      A     DB210.DBX  988.0;
      A     DB210.DBX  982.6;
      S     DB115.DBX   26.4;
      JCN   AFrm;
      L     #ComLine;
      L     128;
      OW    ;
      T     #ComLine;
AFrm: NOP   0;

//Frischwasser
      A     DB1565.DBX   26.1;
      A     #ComU056;
      A     M    103.3;
      =     DB210.DBX  108.0;

      A     DB210.DBX  108.0;
      A     DB210.DBX  102.6;
      S     DB115.DBX   26.4;
      JCN   AXrm;
      L     #ComLine;
      L     256;
      OW    ;
      T     #ComLine;
AXrm: NOP   0;

//Brauhaus
      A     DB1575.DBX   26.1;
      A     #ComU057;
      A     M    103.3;
      =     DB210.DBX  188.0;

      A     DB210.DBX  188.0;
      A     DB210.DBX  182.6;
      S     DB115.DBX   26.4;
      JCN   AYrm;
      L     #ComLine;
      L     512;
      OW    ;
      T     #ComLine;
AYrm: NOP   0;
//Sirupraum
      A     DB1585.DBX   26.1;
      A     #ComU058;
      A     M    103.3;
      =     DB210.DBX  348.0;

      A     DB210.DBX  348.0;
      A     DB210.DBX  342.6;
      S     DB115.DBX   26.4;
      JCN   AZrm;
      L     #ComLine;
      L     1024;
      OW    ;
      T     #ComLine;
AZrm: NOP   0;


      A     #ComSRC;
      A     DB115.DBX  218.4;
      A     M    103.3;
      =     #ReqInlet;

// -------------------------------------------------
// subphase transition
      AN    #reqAnlage;
      AN    DB115.DBX  218.4;
      =     M    103.1;
      JU    COMM;
NETWORK
TITLE =phase 8: Emptying
//SFM   Use                                 Datatype        UoM
//----+-------------------------------------------------------------------------
// 00 : Watch Dog Time                      Duration        min
// 04 : Delay Empty                         Duration        s
// 17 : Level                               Value           l
X8:   SET   ;
// ---------------------------------------------------------------------------
// General CM evaluation
      CALL FC   110 (
           ChkType                  := 3,
           ChkOK                    := #ChkOK);

      AN    #ChkOK;
      S     M    120.3;

// ---------------------------------------------------------------------------
// general functions
      AN    M    121.2;
      A     M    102.3;
      =     #RRel;

      A     M    102.3;
      S     DB115.DBX   26.3;

      A     M    152.1; // Befüllfreigabe
      A     M    102.3;
      S     DB115.DBX   26.0;

// ---------------------------------------------------------------------------
// messages
// ---------------------------------------------------------------------------
// timer & counter

// ---------------------------------------------------------------------------
// pause timer
      ON    M    102.3;
      O     M    150.3;
      S     M    140.3; // Delay Empty

// ---------------------------------------------------------------------------
// communication
      A     DB1435.DBX   26.1;
      A     #ComU043;
      O     ;
      A     DB1455.DBX   26.1;
      A     #ComU045;
      O     ;
      A     DB1475.DBX   26.1;
      A     #ComU047;
      O     ;
      A     DB1485.DBX   26.1;
      A     #ComU048;
      O     ;
      A     DB1495.DBX   26.1;
      A     #ComU049;
      O     ;
      A     DB1505.DBX   26.1;
      A     #ComU050;
      O     ;
      A     DB1515.DBX   26.1;
      A     #ComU051;
      O     ;
      A     DB1525.DBX   26.1;
      A     #ComU052;
      O     ;
      A     DB1545.DBX   26.1;
      A     #ComU054;
      O     ;
      A     DB1555.DBX   26.1;
      A     #ComU055;
      O     ;
      A     DB1565.DBX   26.1;
      A     #ComU056;
      O     ;
      A     DB1575.DBX   26.1;
      A     #ComU057;
      O     ;
      A     DB1585.DBX   26.1;
      A     #ComU058;
      =     #reqAnlage;


// ---------------------------------------------------------------------------
// control modules
      A     M    102.3;

// ---------------------------------------------------------------------------
// transition condition
      A     #U.Seq.User.Bit5; // FILL_REL
      A     DB115.DBX  218.3;
      AN    M    102.2;
      =     M    102.1;
      JCN   N501;
      L     MW   104;
      L     1; // Return to Production
      -I    ;
      T     MW   106;
N501: NOP   0;

      AN    #U.Seq.User.Bit6; // EMPTY_REL
      A     #U.Seq.User.Bit5; // FILL_REL
      AN    M    102.2;
      S     M    102.1;
      JCN   N502;
      L     MW   104;
      L     2; // Return to Filling
      -I    ;
      T     MW   106;
N502: NOP   0;


// ---------------------------------------------------------------------------
// ---------------------------------------------------------------------------
// subphase repeat function
      A     #SubStepMax;
      JCN   Y8;
      L     1;
      T     MW   116;
Y8:   SET   ;

// subphase evaluation
      L     MW   110;
      JL    A800;
      JU    COMM; // subphase  0:
      JU    A801; // subphase  1: Waiting
      JU    A802; // subphase  2: Active
// ---------------------------------------------------------------------------
A800: SET   ;
      S     M    110.7; // Error unknown subphase
      JU    COMM;

// subphase 1: Waiting
A801: SET   ;
      A     M    103.0;
      R     DB115.DBX   26.4;
// -------------------------------------------------
// subphase timer & counter
      A     M    103.0;

// -------------------------------------------------
// subphase actuator
      A     M    103.3;

// -------------------------------------------------
// subphase transition
      A     #reqAnlage;
//      AN    "C01SpiD".LABOR_FREIG_T13.Sig
      =     M    103.1;
      JU    COMM;

// subphase 2: Active
A802: SET   ;
      A     M    103.0;
      =     DB115.DBX   26.4;
// -------------------------------------------------
// subphase timer & counter
      A     M    103.0;

// -------------------------------------------------
// subphase actuator
// Emptying -------------
      CLR   ;
      =     DB115.DBX   26.4;
//KEG
      A     DB1435.DBX   26.1;
      A     #ComU043;
      A     M    103.3;
      =     DB210.DBX  268.0;

      A     DB210.DBX  268.0;
      A     DB210.DBX  262.6;
      S     DB115.DBX   26.4;
      JCN   A3rn;
      L     #ComLine;
      L     1;
      OW    ;
      T     #ComLine;
A3rn: NOP   0;
//A5
      A     DB1455.DBX   26.1;
      A     #ComU045;
      A     M    103.3;
      =     DB210.DBX  828.0;

      A     DB210.DBX  828.0;
      A     DB210.DBX  822.6;
      S     DB115.DBX   26.4;
      JCN   A5rn;
      L     #ComLine;
      L     2;
      OW    ;
      T     #ComLine;
A5rn: NOP   0;

//A7
      A     DB1475.DBX   26.1;
      A     #ComU047;
      A     M    103.3;
      =     DB210.DBX  668.0;

      A     DB210.DBX  668.0;
      A     DB210.DBX  662.6;
      S     DB115.DBX   26.4;
      JCN   A7rn;
      L     #ComLine;
      L     4;
      OW    ;
      T     #ComLine;
A7rn: NOP   0;

//A9
      A     DB1495.DBX   26.1;
      A     #ComU049;
      A     M    103.3;
      =     DB210.DBX  508.0;

      A     DB210.DBX  508.0;
      A     DB210.DBX  502.6;
      S     DB115.DBX   26.4;
      JCN   A9rn;
      L     #ComLine;
      L     8;
      OW    ;
      T     #ComLine;
A9rn: NOP   0;

//A10
      A     DB1505.DBX   26.1;
      A     #ComU050;
      A     M    103.3;
      =     DB210.DBX  428.0;

      A     DB210.DBX  428.0;
      A     DB210.DBX  422.6;
      S     DB115.DBX   26.4;
      JCN   AArn;
      L     #ComLine;
      L     16;
      OW    ;
      T     #ComLine;
AArn: NOP   0;

//A11
      A     DB1515.DBX   26.1;
      A     #ComU051;
      A     M    103.3;
      =     DB210.DBX  908.0;

      A     DB210.DBX  908.0;
      A     DB210.DBX  902.6;
      S     DB115.DBX   26.4;
      JCN   ABrn;
      L     #ComLine;
      L     32;
      OW    ;
      T     #ComLine;
ABrn: NOP   0;

//A12
      A     DB1525.DBX   26.1;
      A     #ComU052;
      A     M    103.3;
      =     DB210.DBX  588.0;

      A     DB210.DBX  588.0;
      A     DB210.DBX  582.6;
      S     DB115.DBX   26.4;
      JCN   ACrn;
      L     #ComLine;
      L     64;
      OW    ;
      T     #ComLine;
ACrn: NOP   0;

//A14
      A     DB1545.DBX   26.1;
      A     #ComU054;
      A     M    103.3;
      =     DB210.DBX  988.0;

      A     DB210.DBX  988.0;
      A     DB210.DBX  982.6;
      S     DB115.DBX   26.4;
      JCN   AFrn;
      L     #ComLine;
      L     128;
      OW    ;
      T     #ComLine;
AFrn: NOP   0;

//Frischwasser
      A     DB1565.DBX   26.1;
      A     #ComU056;
      A     M    103.3;
      =     DB210.DBX  108.0;

      A     DB210.DBX  108.0;
      A     DB210.DBX  102.6;
      S     DB115.DBX   26.4;
      JCN   AXrn;
      L     #ComLine;
      L     256;
      OW    ;
      T     #ComLine;
AXrn: NOP   0;

//Brauhaus
      A     DB1575.DBX   26.1;
      A     #ComU057;
      A     M    103.3;
      =     DB210.DBX  188.0;

      A     DB210.DBX  188.0;
      A     DB210.DBX  182.6;
      S     DB115.DBX   26.4;
      JCN   AYrn;
      L     #ComLine;
      L     512;
      OW    ;
      T     #ComLine;
AYrn: NOP   0;
//Sirupraum
      A     DB1585.DBX   26.1;
      A     #ComU058;
      A     M    103.3;
      =     DB210.DBX  348.0;

      A     DB210.DBX  348.0;
      A     DB210.DBX  342.6;
      S     DB115.DBX   26.4;
      JCN   AZrn;
      L     #ComLine;
      L     1024;
      OW    ;
      T     #ComLine;
AZrn: NOP   0;


// -------------------------------------------------
// subphase transition
      AN    #reqAnlage;
      =     M    103.1;
      JU    COMM;
NETWORK
TITLE =phase 20: Quality Check
//SFM   Use                                 Datatype        UoM
//----+-------------------------------------------------------------------------
// 00 : Watch Dog Time                      Duration        min
// 39 : Q-Status                            Enumeration     min
X20:  SET   ;
// ---------------------------------------------------------------------------
// General CM evaluation
      CALL FC   110 (
           ChkType                  := 3,
           ChkOK                    := #ChkOK);

      AN    #ChkOK;
      S     M    120.3;

// ---------------------------------------------------------------------------
// index evaluation: Q-Status
      CALL FC    45 (
           SFM                      := #U.Seq.SFM[39].Sp,
           Indexes                  := #S2I.SFM39);

// ---------------------------------------------------------------------------
// general functions
      AN    M    121.2;
      A     M    102.3;
      =     #RRel;

// ---------------------------------------------------------------------------
// messages
// ---------------------------------------------------------------------------
// timer & counter
      A     M    102.0;

// ---------------------------------------------------------------------------
// pause timer
// ---------------------------------------------------------------------------
// communication

// ---------------------------------------------------------------------------
// control modules
      A     M    102.3;

// ---------------------------------------------------------------------------
// transition condition
      A     #SubStepMaxD;
      =     M    102.1;

// subphase evaluation
      L     MW   110;
      JL    C000;
      JU    COMM; // subphase  0:
// ---------------------------------------------------------------------------
C000: SET   ;
      S     M    110.7; // Error unknown subphase
      JU    COMM;
NETWORK
TITLE =phase 21: Prepare Tank
//SFM   Use                                 Datatype        UoM
//----+-------------------------------------------------------------------------
// 00 : Watch Dog Time                      Duration        min
// 17 : Level                               Value           l
X21:  SET   ;
// ---------------------------------------------------------------------------
// General CM evaluation
      CALL FC   110 (
           ChkType                  := 3,
           ChkOK                    := #ChkOK);

      AN    #ChkOK;
      S     M    120.3;

// ---------------------------------------------------------------------------
// general functions
      AN    M    121.2;
      A     M    102.3;
      =     #RRel;

// ---------------------------------------------------------------------------
// messages
// ---------------------------------------------------------------------------
// timer & counter
      A     M    102.0;

// ---------------------------------------------------------------------------
// pause timer
// ---------------------------------------------------------------------------
// communication

// ---------------------------------------------------------------------------
// control modules

      CLR   ;
      =     DB211.DBX  503.1; // Filling Hand Valve
      =     DB211.DBX  623.1; // CIP Hand Valve

      A     M    102.3;
      =     DB211.DBX  503.0; // Filling Hand Valve
      =     DB211.DBX  623.0; // CIP Hand Valve

// ---------------------------------------------------------------------------
// transition condition
      AN    DB211.DBX  498.7; // Filling Hand Valve
      AN    DB211.DBX  618.7; // CIP Hand Valve
      AN    M    102.2;
      =     M    102.1;

// subphase evaluation
      L     MW   110;
      JL    C100;
      JU    COMM; // subphase  0:
// ---------------------------------------------------------------------------
C100: SET   ;
      S     M    110.7; // Error unknown subphase
      JU    COMM;
NETWORK
TITLE =phase 23: Connect Tank
//SFM   Use                                 Datatype        UoM
//----+-------------------------------------------------------------------------
// 00 : Watch Dog Time                      Duration        min
X23:  SET   ;
// ---------------------------------------------------------------------------
// General CM evaluation
      CALL FC   110 (
           ChkType                  := 3,
           ChkOK                    := #ChkOK);

      AN    #ChkOK;
      S     M    120.3;

// ---------------------------------------------------------------------------
// general functions
      AN    M    121.2;
      A     M    102.3;
      =     #RRel;

// ---------------------------------------------------------------------------
// messages
// ---------------------------------------------------------------------------
// timer & counter
      A     M    102.0;

// ---------------------------------------------------------------------------
// pause timer
// ---------------------------------------------------------------------------
// communication

// ---------------------------------------------------------------------------
// control modules
      A     M    102.3;

// ---------------------------------------------------------------------------
// transition condition
      A     #SubStepMaxD;
      =     M    102.1;

// subphase evaluation
      L     MW   110;
      JL    C300;
      JU    COMM; // subphase  0:
// ---------------------------------------------------------------------------
C300: SET   ;
      S     M    110.7; // Error unknown subphase
      JU    COMM;
NETWORK
TITLE =phase 31: CIP Start
//SFM   Use                                 Datatype        UoM
//----+-------------------------------------------------------------------------
// 00 : Watch Dog Time                      Duration        min
X31:  SET   ;
// ---------------------------------------------------------------------------
// General CM evaluation
      CALL FC   110 (
           ChkType                  := 4,
           ChkOK                    := #ChkOK);

      AN    #ChkOK;
      S     M    120.3;

// ---------------------------------------------------------------------------
// general functions
      AN    M    121.2;
      A     M    102.3;
      =     #RRel;

// ---------------------------------------------------------------------------
// messages
// ---------------------------------------------------------------------------
// timer & counter
// ---------------------------------------------------------------------------
// pause timer
// ---------------------------------------------------------------------------
// communication

// ---------------------------------------------------------------------------
// control modules

// ---------------------------------------------------------------------------
// transition condition
      A     #SubStepMaxD;
      =     M    102.1;

// ---------------------------------------------------------------------------
// ---------------------------------------------------------------------------
// subphase repeat function
//      A     #SubStepMax
//      JCN  Y31
//      L     1
//      T     "SOSubStepNew"
//Y31:  SET

// subphase evaluation
      L     MW   110;
      JL    D100;
      JU    COMM; // subphase  0:
      JU    D101; // subphase  1: Wait For CIP
      JU    D102; // subphase  2: Wait For Partner
// ---------------------------------------------------------------------------
D100: SET   ;
      S     M    110.7; // Error unknown subphase
      JU    COMM;

// subphase 1: Wait For CIP
D101: SET   ;

// -------------------------------------------------
// CIP Signals ---
// Start Signal
      A     M    120.0;
      A     M    103.3;
      =     DB115.DBX  172.4;
      JCN   CIPS;
      L     MD   124;
      T     DB502.DBD    0;
      T     DB502.DBD  156;
CIPS: NOP   0;

// -------------------------------------------------
// subphase actuator

// -------------------------------------------------
// subphase transition
// CIP Ready
      A     #ComCIP;
      A     DB115.DBX  123.5;
      A     DB115.DBX  120.0;
// CIP Distribution Ready
      A     #ComCIPDist;
      A     DB1945.DBX   27.5;
      A     DB1945.DBX   24.0;
      =     M    103.1;
      JU    COMM;

// subphase 2: Wait For Partner
D102: SET   ;

// -------------------------------------------------
// subphase timer & counter
      A     M    103.0;

// -------------------------------------------------
// subphase actuator
      A     M    103.3;

// -------------------------------------------------
// subphase transition
      CLR   ;
      =     M    103.1;
      JU    COMM;
NETWORK
TITLE =phase 32: CIP Prerun
//SFM   Use                                 Datatype        UoM
//----+-------------------------------------------------------------------------
// 00 : Watch Dog Time                      Duration        min
// 01 : Step Time                           Duration        min
// 04 : Delay Level                         Duration        s
// 15 : Amount                              Value           m3
// 17 : Level                               Value           l
// 22 : Agitator Speed                      Value           %
// 27 : CIP Prerun                          Enumeration     min
// 28 : CIP Return                          Enumeration     min
// 29 : CIP Pump Speed                      Value           %
// 34 : CIP Prerun Flow                     Value           m3/h
// 35 : CIP Prerun Pressure                 Value           bar
// 37 : CIP Pump Mode                       Enumeration     min
X32:  SET   ;
// ---------------------------------------------------------------------------
// General CM evaluation
      CALL FC   110 (
           ChkType                  := 4,
           ChkOK                    := #ChkOK);

      AN    #ChkOK;
      S     M    120.3;

// ---------------------------------------------------------------------------
// index evaluation: CIP Prerun
      CALL FC    45 (
           SFM                      := #U.Seq.SFM[27].Sp,
           Indexes                  := #S2I.SFM27);

// ---------------------------------------------------------------------------
// index evaluation: CIP Return
      CALL FC    45 (
           SFM                      := #U.Seq.SFM[28].Sp,
           Indexes                  := #S2I.SFM28);

// ---------------------------------------------------------------------------
// index evaluation: CIP Pump Mode
      CALL FC    45 (
           SFM                      := #U.Seq.SFM[37].Sp,
           Indexes                  := #S2I.SFM37);

// ---------------------------------------------------------------------------
// general functions
      AN    M    121.2;
      A     M    102.3;
      =     #RRel;

// ---------------------------------------------------------------------------
// messages
// CIP Unit
      AN    #ComCIP;
      ON    DB115.DBX  123.4;
      ON    DB115.DBX  123.5;
      JCN   x321;
      R     #RRel;
      L     949; // CIP Not Ready!
      T     MD    90;
x321: NOP   0;

// CIP Distribution Unit
      AN    #ComCIPDist;
      ON    DB1945.DBX   27.4;
      ON    DB1945.DBX   27.5;
      JCN   x322;
      R     #RRel;
      L     949; // CIP Partner Not Ready!
      T     MD    90;
x322: NOP   0;

// CIP Signals ---
      L     #U.Seq.SFM[17].Sp;
      L     0.000000e+000;
      <=R   ;
      O     M    152.0;
      =     #xTmp;
      CALL FC   716 (
           StepOnSFMSP              := #U.Seq.SFM[26].Sp,
           EmptySig                 := DB211.DBX   78.7,
           EmptyLevel               := #xTmp,
           CIPPumpRun               := DB115.DBX  124.3,
           CIPReady                 := DB115.DBX  123.5,
           Empty                    := DB115.DBX   26.5,
           TransCondOK              := M    102.1,
           RRel                     := #RRel);

// ---------------------------------------------------------------------------
// timer & counter
// Done in "CIPUnitC"

// ---------------------------------------------------------------------------
// communication
// Active, Prerun & Return
      A     M    102.0;
      =     DB115.DBX  171.4;
      =     DB115.DBX  172.6;
      =     DB115.DBX  172.7;

// Run Release
      A     #RRel;
      =     DB115.DBX  171.5;

// Prerun Pump
      A     DB115.DBX  172.6;
      AN    #S2I.SFM37.I00;
      A     #RRel;
      =     DB115.DBX  173.3;

// Return Pump
      AN    DB115.DBX   26.5;
      A     #RRel;
      =     DB115.DBX  173.4;

// ---------------------------------------------------------------------------
// control modules (Own CM's)
      A     M    102.0;
      =     DB210.DBX 1228.0;
      =     DB210.DBX 2268.0;

      A     M    102.3;
      =     DB210.DBX 1148.0;

// ---------------------------------------------------------------------------
// transition condition
//      A     #SubStepMaxD
//      =     "SOPD"

// subphase evaluation
      L     MW   110;
      JL    D200;
      JU    COMM; // subphase  0:
// ---------------------------------------------------------------------------
D200: SET   ;
      S     M    110.7; // Error unknown subphase
      JU    COMM;
NETWORK
TITLE =phase 33: CIP Return
//SFM   Use                                 Datatype        UoM
//----+-------------------------------------------------------------------------
// 00 : Watch Dog Time                      Duration        min
// 01 : Step Time                           Duration        min
// 04 : Delay Level                         Duration        s
// 06 : Delay Switchpoint                   Duration        s
// 15 : Amount                              Value           m3
// 17 : Level                               Value           l
// 22 : Agitator Speed                      Value           %
// 26 : CIP Step On Condition               Enumeration     min
// 27 : CIP Prerun                          Enumeration     min
// 28 : CIP Return                          Enumeration     min
// 29 : CIP Pump Speed                      Value           %
// 30 : CIP Return Temperature              Value           °C
// 32 : CIP Return Conductivity             Value           mS
// 34 : CIP Prerun Flow                     Value           m3/h
// 35 : CIP Prerun Pressure                 Value           bar
// 37 : CIP Pump Mode                       Enumeration     min
X33:  SET   ;
// ---------------------------------------------------------------------------
// General CM evaluation
      CALL FC   110 (
           ChkType                  := 4,
           ChkOK                    := #ChkOK);

      AN    #ChkOK;
      S     M    120.3;

// ---------------------------------------------------------------------------
// index evaluation: CIP Step On Condition
      CALL FC    45 (
           SFM                      := #U.Seq.SFM[26].Sp,
           Indexes                  := #S2I.SFM26);

// ---------------------------------------------------------------------------
// index evaluation: CIP Prerun
      CALL FC    45 (
           SFM                      := #U.Seq.SFM[27].Sp,
           Indexes                  := #S2I.SFM27);

// ---------------------------------------------------------------------------
// index evaluation: CIP Return
      CALL FC    45 (
           SFM                      := #U.Seq.SFM[28].Sp,
           Indexes                  := #S2I.SFM28);

// ---------------------------------------------------------------------------
// index evaluation: CIP Pump Mode
      CALL FC    45 (
           SFM                      := #U.Seq.SFM[37].Sp,
           Indexes                  := #S2I.SFM37);

// ---------------------------------------------------------------------------
// general functions
      AN    M    121.2;
      A     M    102.3;
      =     #RRel;

// ---------------------------------------------------------------------------
// messages
// CIP Unit
      AN    #ComCIP;
      ON    DB115.DBX  123.4;
      ON    DB115.DBX  123.5;
      JCN   x331;
      R     #RRel;
      L     949; // CIP Not Ready!
      T     MD    90;
x331: NOP   0;

// CIP Distribution Unit
      AN    #ComCIPDist;
      ON    DB1945.DBX   27.4;
      ON    DB1945.DBX   27.5;
      JCN   x332;
      R     #RRel;
      L     949; // CIP Partner Not Ready!
      T     MD    90;
x332: NOP   0;

// CIP Signals ---
      L     #U.Seq.SFM[17].Sp;
      L     0.000000e+000;
      <=R   ;
      O     M    152.0;
      =     #xTmp;

      CALL FC   716 (
           StepOnSFMSP              := #U.Seq.SFM[26].Sp,
           EmptySig                 := DB211.DBX   78.7,
           EmptyLevel               := #xTmp,
           CIPPumpRun               := DB115.DBX  124.3,
           CIPReady                 := DB115.DBX  123.5,
           Empty                    := #Empty,
           TransCondOK              := M    102.1,
           RRel                     := #RRel);

// ---------------------------------------------------------------------------
// timer & counter
// Done in "CIPUnitC"

// ---------------------------------------------------------------------------
// communication
// Active, Prerun & Return
      A     M    102.0;
      =     DB115.DBX  171.4;
      =     DB115.DBX  172.6;
      =     DB115.DBX  172.7;

// Run Release
      A     #RRel;
      =     DB115.DBX  171.5;

// Prerun Pump
      A     DB115.DBX  172.6;
      AN    #S2I.SFM37.I00;
      A     #RRel;
      =     DB115.DBX  173.3;

// Return Pump
      AN    #Empty;
      A     #RRel;
      =     DB115.DBX  173.4;

// Bypass Valve
      A     M    102.3;
      =     DB115.DBX  173.5;

// ---------------------------------------------------------------------------
// control modules (Own CM's)
      A     M    102.0;
      =     DB210.DBX 2268.0;

// Bypass Valve Used in CIP Distribution
//      A     "SOPA"
//      =     "C01ActD".RV1_T13.ACo

//      A     "SOPH"
//      =     "C01ActD".T13_RR1.ACo

// ---------------------------------------------------------------------------
// transition condition
//      A     #SubStepMaxD
//      =     "SOPD"

// subphase evaluation
      L     MW   110;
      JL    D300;
      JU    COMM; // subphase  0:
// ---------------------------------------------------------------------------
D300: SET   ;
      S     M    110.7; // Error unknown subphase
      JU    COMM;
NETWORK
TITLE =phase 34: CIP Rinsing
//SFM   Use                                 Datatype        UoM
//----+-------------------------------------------------------------------------
// 00 : Watch Dog Time                      Duration        min
// 01 : Step Time                           Duration        min
// 04 : Delay Level                         Duration        s
// 05 : Substep Time                        Duration        s
// 06 : Delay Switchpoint                   Duration        s
// 15 : Amount                              Value           m3
// 17 : Level                               Value           l
// 22 : Agitator Speed                      Value           %
// 27 : CIP Prerun                          Enumeration     min
// 28 : CIP Return                          Enumeration     min
// 29 : CIP Pump Speed                      Value           %
// 30 : CIP Return Temperature              Value           °C
// 32 : CIP Return Conductivity             Value           mS
// 34 : CIP Prerun Flow                     Value           m3/h
// 35 : CIP Prerun Pressure                 Value           bar
// 37 : CIP Pump Mode                       Enumeration     min
// 59 : Interval Counter                    Value           No.
X34:  SET   ;
// ---------------------------------------------------------------------------
// General CM evaluation
      CALL FC   110 (
           ChkType                  := 4,
           ChkOK                    := #ChkOK);

      AN    #ChkOK;
      S     M    120.3;

// ---------------------------------------------------------------------------
// index evaluation: CIP Prerun
      CALL FC    45 (
           SFM                      := #U.Seq.SFM[27].Sp,
           Indexes                  := #S2I.SFM27);

// ---------------------------------------------------------------------------
// index evaluation: CIP Return
      CALL FC    45 (
           SFM                      := #U.Seq.SFM[28].Sp,
           Indexes                  := #S2I.SFM28);

// ---------------------------------------------------------------------------
// index evaluation: CIP Pump Mode
      CALL FC    45 (
           SFM                      := #U.Seq.SFM[37].Sp,
           Indexes                  := #S2I.SFM37);

// ---------------------------------------------------------------------------
// general functions
      AN    M    121.2;
      A     M    102.3;
      =     #RRel;

// ---------------------------------------------------------------------------
// messages
// CIP Unit
      AN    #ComCIP;
      ON    DB115.DBX  123.4;
      ON    DB115.DBX  123.5;
      JCN   x341;
      R     #RRel;
      L     949; // CIP Not Ready!
      T     MD    90;
x341: NOP   0;

// CIP Distribution Unit
      AN    #ComCIPDist;
      ON    DB1945.DBX   27.4;
      ON    DB1945.DBX   27.5;
      JCN   x342;
      R     #RRel;
      L     949; // CIP Partner Not Ready!
      T     MD    90;
x342: NOP   0;

// CIP Signals ---
      L     #U.Seq.SFM[17].Sp;
      L     0.000000e+000;
      <=R   ;
      O     M    152.0;
      =     #xTmp;

      CALL FC   716 (
           StepOnSFMSP              := #U.Seq.SFM[26].Sp,
           EmptySig                 := DB211.DBX   78.7,
           EmptyLevel               := #xTmp,
           CIPPumpRun               := DB115.DBX  124.3,
           CIPReady                 := DB115.DBX  123.5,
           Empty                    := DB115.DBX   26.5,
           TransCondOK              := M    102.1,
           RRel                     := #RRel);

// ---------------------------------------------------------------------------
// timer & counter
// Done in "CIPUnitC"

// ---------------------------------------------------------------------------
// communication
// Active, Prerun & Return
      A     M    102.0;
      =     DB115.DBX  171.4;
      =     DB115.DBX  172.6;
      =     DB115.DBX  172.7;

// Run Release
      A     #RRel;
      =     DB115.DBX  171.5;

// Prerun Pump
      A     DB115.DBX  172.6;
      AN    #S2I.SFM37.I00;
      A     #RRel;
      =     DB115.DBX  173.3;

// Return Pump
      AN    DB115.DBX   26.5;
      A     #RRel;
      =     DB115.DBX  173.4;

// ---------------------------------------------------------------------------
// control modules (Own CM's)
      A     M    102.0;
      =     DB210.DBX 1228.0;
      =     DB210.DBX 2268.0;

      A     M    102.3;
      =     DB210.DBX 1148.0;

// ---------------------------------------------------------------------------
// transition condition (Check CIPUnitC)
//      A     #SubStepMaxD
//      =     "SOPD"

// ---------------------------------------------------------------------------
// ---------------------------------------------------------------------------
// subphase repeat function
      A     #SubStepMax;
      JCN   Y34;
      L     1;
      T     MW   116;
Y34:  NOP   0;

      A     #SubStepMax;
      AN    M    103.0;
      JCN   Y34a;
      L     #U.Seq.SFM[59].Val; // Increment Interval Counter
      L     1.000000e+000;
      +R    ;
      T     #U.Seq.SFM[59].Val;
Y34a: SET   ;
      A     M    102.2;
      ON    M    102.0;
      JCN   IntR; // Reset Interval Counter at Start and End Of Phase
      L     0.000000e+000;
      T     #U.Seq.SFM[59].Val;
IntR: NOP   0;

// subphase evaluation
      L     MW   110;
      JL    D400;
      JU    COMM; // subphase  0:
      JU    D401; // subphase  1: Pause
      JU    D402; // subphase  2: Main
      JU    D403; // subphase  3: Expulse
      JU    D404; // subphase  4: Seat Lift
      JU    D400; // subphase  5:
      JU    D406; // subphase  6: Shaft Rinse
      JU    D407; // subphase  7: Drain
// ---------------------------------------------------------------------------
D400: SET   ;
      S     M    110.7; // Error unknown subphase
      JU    COMM;

// subphase 1: Pause
D401: SET   ;
      A     M    103.0;
      R     DB115.DBX  173.3;

// -------------------------------------------------
// subphase timer & counter
      A     M    103.0;
      =     M    130.4; // Substep Time

// -------------------------------------------------
// subphase actuator

// -------------------------------------------------
// subphase transition
      A     M    150.3; // Delay Level
      A     M    130.3;
      O     M    150.4; // Substep Time Done
      =     M    103.1;
      JU    COMM;

// subphase 2: Main
D402: SET   ;

// -------------------------------------------------
// subphase timer & counter
      A     M    103.0;
      =     M    130.4; // Substep Time

// -------------------------------------------------
// subphase actuator
      A     M    103.3;

// -------------------------------------------------
// subphase transition
      A     M    150.4; // Substep Time Done
      =     M    103.1;
      JU    COMM;

// subphase 3: Expulse
D403: SET   ;

// -------------------------------------------------
// subphase timer & counter
      A     M    103.0;

// -------------------------------------------------
// subphase actuator
      A     M    103.3;

// -------------------------------------------------
// subphase transition
      CLR   ;
      =     M    103.1;
      JU    COMM;

// subphase 4: Seat Lift
D404: SET   ;

// -------------------------------------------------
// subphase timer & counter
      A     M    103.0;

// -------------------------------------------------
// subphase actuator
      A     M    103.3;

// -------------------------------------------------
// subphase transition
      CLR   ;
      =     M    103.1;
      JU    COMM;

// subphase 6: Shaft Rinse
D406: SET   ;

// -------------------------------------------------
// subphase timer & counter
      A     M    103.0;

// -------------------------------------------------
// subphase actuator
      A     M    103.3;

// -------------------------------------------------
// subphase transition
      CLR   ;
      =     M    103.1;
      JU    COMM;

// subphase 7: Drain
D407: SET   ;

// -------------------------------------------------
// subphase timer & counter
      A     M    103.0;

// -------------------------------------------------
// subphase actuator
      A     M    103.3;

// -------------------------------------------------
// subphase transition
      CLR   ;
      =     M    103.1;
      JU    COMM;
NETWORK
TITLE =phase 35: CIP Emptying
//SFM   Use                                 Datatype        UoM
//----+-------------------------------------------------------------------------
// 00 : Watch Dog Time                      Duration        min
// 04 : Delay Empty                         Duration        s
// 17 : Level                               Value           l
// 22 : Agitator Speed                      Value           %
// 26 : Step On Empty                       Enumeration     min
// 28 : CIP Return                          Enumeration     min
X35:  SET   ;
// ---------------------------------------------------------------------------
// General CM evaluation
      CALL FC   110 (
           ChkType                  := 4,
           ChkOK                    := #ChkOK);

      AN    #ChkOK;
      S     M    120.3;

// ---------------------------------------------------------------------------
// index evaluation: Step On Empty
      CALL FC    45 (
           SFM                      := #U.Seq.SFM[26].Sp,
           Indexes                  := #S2I.SFM26);

// ---------------------------------------------------------------------------
// index evaluation: CIP Return
      CALL FC    45 (
           SFM                      := #U.Seq.SFM[28].Sp,
           Indexes                  := #S2I.SFM28);

// ---------------------------------------------------------------------------
// general functions
      AN    M    121.2;
      A     M    102.3;
      =     #RRel;

// ---------------------------------------------------------------------------
// messages
// CIP Unit
      AN    #ComCIP;
      ON    DB115.DBX  123.4;
      ON    DB115.DBX  123.5;
      JCN   x351;
      R     #RRel;
      L     949; // CIP Not Ready!
      T     MD    90;
x351: NOP   0;

// CIP Distribution Unit
      AN    #ComCIPDist;
      ON    DB1945.DBX   27.4;
      ON    DB1945.DBX   27.5;
      JCN   x352;
      R     #RRel;
      L     949; // CIP Partner Not Ready!
      T     MD    90;
x352: NOP   0;

// CIP Signals ---
      CALL FC   716 (
           StepOnSFMSP              := #U.Seq.SFM[26].Sp,
           EmptySig                 := DB211.DBX   78.7,
           EmptyLevel               := M    152.0,
           CIPPumpRun               := DB115.DBX  124.3,
           CIPReady                 := DB115.DBX  123.5,
           Empty                    := DB115.DBX   26.5,
           TransCondOK              := M    102.1,
           RRel                     := #RRel);

// ---------------------------------------------------------------------------
// timer & counter
// Done in "CIPUnitC"

// ---------------------------------------------------------------------------
// communication
// Active, Prerun & Return
      A     M    102.0;
      =     DB115.DBX  171.4;
      =     DB115.DBX  172.7;

// Run Release
      A     #RRel;
      =     DB115.DBX  171.5;

// Prerun Pump
      A     DB115.DBX  172.6;
      AN    #S2I.SFM37.I00;
      A     #RRel;
      CLR   ;
      =     DB115.DBX  173.3;

// Return Pump
      AN    DB115.DBX   26.5;
      A     #RRel;
      =     DB115.DBX  173.4;

// ---------------------------------------------------------------------------
// control modules (Own CM's)
      A     M    102.0;
      =     DB210.DBX 1228.0;
      =     DB210.DBX 2268.0;

      A     M    102.3;
      =     DB210.DBX 1148.0;

// ---------------------------------------------------------------------------
// transition condition
//      A     #SubStepMaxD
//      =     "SOPD"


// subphase evaluation
      L     MW   110;
      JL    D500;
      JU    COMM; // subphase  0:
// ---------------------------------------------------------------------------
D500: SET   ;
      S     M    110.7; // Error unknown subphase
      JU    COMM;
NETWORK
TITLE =phase 36: CIP Drain
//SFM   Use                                 Datatype        UoM
//----+-------------------------------------------------------------------------
// 00 : Watch Dog Time                      Duration        Min
// 04 : Delay Empty                         Duration        #sec
X36:  SET   ;
// ---------------------------------------------------------------------------
// General CM evaluation
      CALL FC   110 (
           ChkType                  := 4,
           ChkOK                    := #ChkOK);

      AN    #ChkOK;
      S     M    120.3;

// ---------------------------------------------------------------------------
// general functions
      AN    M    121.2;
      A     M    102.3;
      =     #RRel;

// ---------------------------------------------------------------------------
// messages
// ---------------------------------------------------------------------------
// timer & counter
      A     M    102.0;

// ---------------------------------------------------------------------------
// pause timer
      ON    M    102.3;
      O     M    150.3;
      S     M    140.3; // Delay Empty

// ---------------------------------------------------------------------------
// communication

// ---------------------------------------------------------------------------
// control modules
      A     M    102.3;

// ---------------------------------------------------------------------------
// transition condition
      A     #SubStepMaxD;
      =     M    102.1;

// subphase evaluation
      L     MW   110;
      JL    D600;
      JU    COMM; // subphase  0:
// ---------------------------------------------------------------------------
D600: SET   ;
      S     M    110.7; // Error unknown subphase
      JU    COMM;
NETWORK
TITLE =phase 40: CIP End
//SFM   Use                                 Datatype        UoM
//----+-------------------------------------------------------------------------
// 00 : Watch Dog Time                      Duration        min
X40:  SET   ;
// ---------------------------------------------------------------------------
// General CM evaluation
      CALL FC   110 (
           ChkType                  := 4,
           ChkOK                    := #ChkOK);

      AN    #ChkOK;
      S     M    120.3;
// ---------------------------------------------------------------------------
// general functions
//      AN    "SOSTAl"
      A     M    102.3;
      =     #RRel;

// CIP Signals ---
      CALL FC   716 (
           StepOnSFMSP              := 0.000000e+000,
           EmptySig                 := FALSE,
           EmptyLevel               := FALSE,
           CIPPumpRun               := FALSE,
           CIPReady                 := FALSE,
           Empty                    := #xTmp,
           TransCondOK              := #xTmp,
           RRel                     := #RRel);

// ---------------------------------------------------------------------------
// communication
      A     M    102.0;
      =     DB115.DBX  173.7;

// ---------------------------------------------------------------------------
// transition condition
      AN    #ComCIP;
      AN    #ComCIPDist;
      =     M    102.1;

// subphase evaluation
      L     MW   110;
      JL    E000;
      JU    COMM; // subphase  0:
// ---------------------------------------------------------------------------
E000: SET   ;
      S     M    110.7; // Error unknown subphase
      JU    COMM;

NETWORK
TITLE =End Of Sequence Organisation
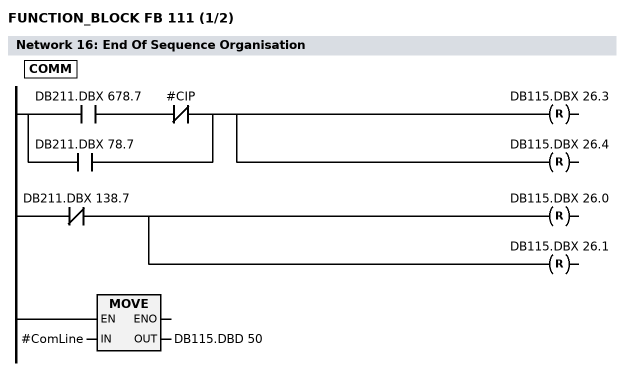

COMM: SET   ;

// ---------------------------------------------------------------------------
// pause timer unit parameter

// Laborfreigabe
      A     DB211.DBX  678.7;
      AN    #CIP;
      O     DB211.DBX   78.7;
      R     DB115.DBX   26.3;
      R     DB115.DBX   26.4;

      AN    DB211.DBX  138.7;
      R     DB115.DBX   26.0;
      R     DB115.DBX   26.1;

// Line Communication
      L     #ComLine;
      T     DB115.DBD   50;

NETWORK
TITLE =General Post Phase Controls
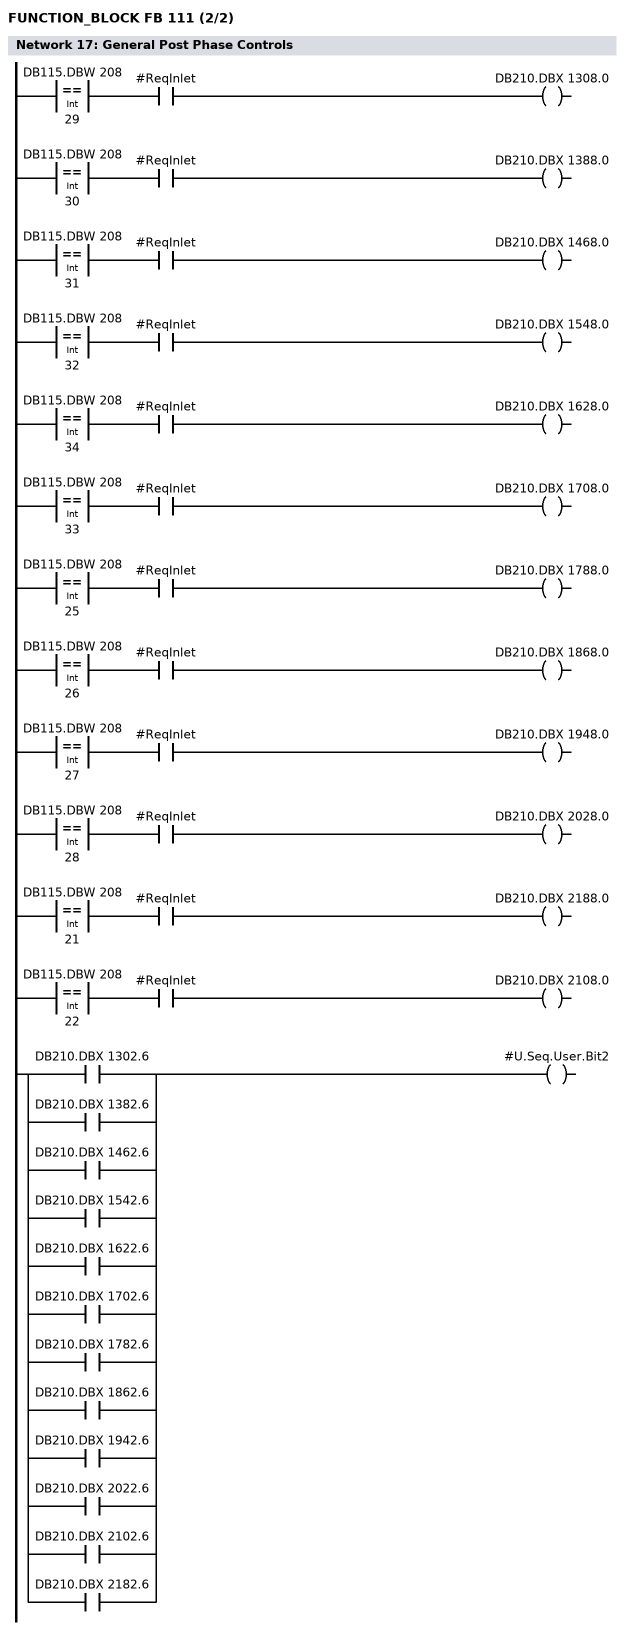

      NOP   0;

// ---------------------------------------------------------------------------
// general postphase controls
// Inlet Control
      L     DB115.DBW  208;
      L     29; // B6F
      ==I   ;
      A     #ReqInlet;
      =     DB210.DBX 1308.0;

      L     DB115.DBW  208;
      L     30; // H6
      ==I   ;
      A     #ReqInlet;
      =     DB210.DBX 1388.0;

      L     DB115.DBW  208;
      L     31; // J6
      ==I   ;
      A     #ReqInlet;
      =     DB210.DBX 1468.0;

      L     DB115.DBW  208;
      L     32; // L6F
      ==I   ;
      A     #ReqInlet;
      =     DB210.DBX 1548.0;

      L     DB115.DBW  208;
      L     34; // D6
      ==I   ;
      A     #ReqInlet;
      =     DB210.DBX 1628.0;

      L     DB115.DBW  208;
      L     33; // B6
      ==I   ;
      A     #ReqInlet;
      =     DB210.DBX 1708.0;

      L     DB115.DBW  208;
      L     25; // A
      ==I   ;
      A     #ReqInlet;
      =     DB210.DBX 1788.0;

      L     DB115.DBW  208;
      L     26; // B
      ==I   ;
      A     #ReqInlet;
      =     DB210.DBX 1868.0;

      L     DB115.DBW  208;
      L     27; //CF
      ==I   ;
      A     #ReqInlet;
      =     DB210.DBX 1948.0;

      L     DB115.DBW  208;
      L     28; // C1
      ==I   ;
      A     #ReqInlet;
      =     DB210.DBX 2028.0;

      L     DB115.DBW  208;
      L     21; // VE1
      ==I   ;
      A     #ReqInlet;
      =     DB210.DBX 2188.0;

      L     DB115.DBW  208;
      L     22; // VE2
      ==I   ;
      A     #ReqInlet;
      =     DB210.DBX 2108.0;

      A     DB210.DBX 1302.6;
      O     DB210.DBX 1382.6;
      O     DB210.DBX 1462.6;
      O     DB210.DBX 1542.6;
      O     DB210.DBX 1622.6;
      O     DB210.DBX 1702.6;
      O     DB210.DBX 1782.6;
      O     DB210.DBX 1862.6;
      O     DB210.DBX 1942.6;
      O     DB210.DBX 2022.6;
      O     DB210.DBX 2102.6;
      O     DB210.DBX 2182.6;
      =     #U.Seq.User.Bit2;

NETWORK
TITLE =Process Status Management

      NOP   0;
// ---------------------------------------------------------------------------
// Signal Control
      OPN   DB   500;
      L     #UnitNo;
      L     32; //U Structure Length
      *I    ;
      L     20; //DB Heading Offset
      +I    ;
      SLD   3;
      LAR2  ;

// -------------------------------------------------
// Maintenance
      A     #U.Seq.Switch.Sw31;
      OPN   DB   500;
      =     DBX [AR2,P#0.0]; //"PStatD".U[#UnitNo].MTNC
// -------------------------------------------------
// CIP Required
// -------------------------------------------------
// CIP Active
// -------------------------------------------------
// CIP Clean
// -------------------------------------------------
// SIP Required
// -------------------------------------------------
// SIP Active
// -------------------------------------------------
// SIP Clean
// -------------------------------------------------
// Full
      A     DB115.DBX   26.2;
      OPN   DB   500;
      =     DBX [AR2,P#0.7]; //"PStatD".U[#UnitNo].FULL
// -------------------------------------------------
// Filling
      A     DB115.DBX   26.1;
      OPN   DB   500;
      =     DBX [AR2,P#1.0]; //"PStatD".U[#UnitNo].FILL
// -------------------------------------------------
// Ready For Filling
      A     DB115.DBX   26.0;
      OPN   DB   500;
      =     DBX [AR2,P#1.1]; //"PStatD".U[#UnitNo].RFFI
// -------------------------------------------------
// Empty
      A     DB115.DBX   26.5;
      OPN   DB   500;
      =     DBX [AR2,P#1.2]; //"PStatD".U[#UnitNo].EMTY
// -------------------------------------------------
// Emptying
      A     DB115.DBX   26.4;
      OPN   DB   500;
      =     DBX [AR2,P#1.3]; //"PStatD".U[#UnitNo].EMTI
// -------------------------------------------------
// Ready For Emptying
      A     DB115.DBX   26.3;
      OPN   DB   500;
      =     DBX [AR2,P#1.4]; //"PStatD".U[#UnitNo].RFEM
// -------------------------------------------------
// Reserved
//      A     #ComXYZ
//      OPN   "PStatD"
//      =     DBX [AR2,P#1.5]             //"PStatD".U[#UnitNo].RESV
// -------------------------------------------------
// Production
// -------------------------------------------------
// Used

// -------------------------------------------------
// PStat Function Call

      CALL FC   500 (
           UnitNo                   := #UnitNo,
           PStatModVal              := DB215.DBD  234);


NETWORK
TITLE =Unit Hold Request and Messages

      SET   ;

// ---------------------------------------------------------------------------
// Set unit to "hold" if maintenance
      AN    #U.Seq.Switch.Sw31; // maintenance !
      JC    NCO1;
      S     M    120.3;
      L     998; // "Unit in maintenance !"
      T     MD    90;

// ---------------------------------------------------------------------------
// Set unit to "hold" if emergency stop
NCO1: A     #EStopOK;
      JC    NCO2;
      S     M    120.3;
      L     999; // "Emergency stop !"
      T     MD    90;
NCO2: NOP   0;

END_FUNCTION_BLOCK

FUNCTION_BLOCK FB 113
TITLE =C01: Water Tank x
AUTHOR : Woermann
FAMILY : BOTEC_F1
NAME : C01E
VERSION : 1.2
CODE_VERSION1


VAR
  U : UDT 111;
END_VAR
VAR_TEMP
  CIP : BOOL ;	//CIP active
  UNIM : BOOL ;	//Unit Not In Maintenance
  GenRel : BOOL ;	//general OK (emergency and maintenance OK)
  EStopOK : BOOL ;	//emergency OK
  UnitNo : INT ;	//unit number
  xTmp : BOOL ;	//Temporary Bool
  iTmp : INT ;	//Temporary INT
  rTmp : REAL ;	//Temporary REAL
  dTmp : DINT ;	//Temporary DINT (free for general use)
  RetValInt : INT ;	//return value
  ComCIP1 : BOOL ;	//CIP1 in use
  ComCIP3 : BOOL ;	//CIP3 in use
  LabRel : BOOL ;	//Laborfreigabe
END_VAR
BEGIN
NETWORK
TITLE =General


      SET   ;
// Simulation ---------------------------------------------------------------
      A     #U.Seq.User.Bit63;
      CC    FB   119;
      A     #U.Seq.Sim;
      =     #U.Seq.User.Bit63; //Help bit for simulation

// get unit number ----------------------------------------------------------
      L     MB   112;
      T     #UnitNo;

// CIP ----------------------------------------------------------------------
      L     #U.Seq.ProgNo;
      L     0;
      <D    ;
      =     #CIP;

// emergency OK -------------------------------------------------------------
      A     DB115.DBX   27.0; //Emergency Stop OK
      =     #EStopOK;

// Write Unit in Maintenance ------------------------------------------------

      AN    #U.Seq.Switch.Sw31;
      =     #UNIM;

// emergency and maintenance OK ---------------------------------------------
      A     #EStopOK;
      A     #UNIM;
      =     #GenRel;

// communication ------------------------------------------------------------
      UC    FB   115;

NETWORK
TITLE =Analog Inputs

      NOP   0;

// ----------------------------------------------------------
// LI_T13 Niveau Tank 13
// ----------------------------------------------------------
      L     #U.Seq.SFM[63].Sp; // !!! insert correct SFM !!!
      T     DB213.DBD  238;

//      CLR
//      =     "C01AniD".LI_T13.EAlHH

NETWORK
TITLE =Universal Value

      NOP   0;

// ----------------------------------------------------------
// unv001 Process Status
// ----------------------------------------------------------
// process value to UnV
//      L     0.000000e+000
//      T     "C01UnVD".unv001.ValExt

// ----------------------------------------------------------
// unv002 Universal Value 02
// ----------------------------------------------------------
// process value to UnV
//      L     0.000000e+000
//      T     "C01UnVD".unv002.ValExt

      A     M    101.3;
      JCN   STG1;
      L     DB213.DBD  146;
      L     #U.Seq.User.Real11;
      -R    ;
      L     6.000000e+002;
      *R    ;
      T     #rTmp;
      L     DB215.DBD  362;
      L     1.000000e+002;
      *R    ;
      L     #rTmp;
      +R    ;
      L     1.010000e+002;
      /R    ;
      JO    STG1;
      T     DB215.DBD  362;
      L     DB213.DBD  146;
      T     #U.Seq.User.Real11;
STG1: NOP   0;

// ----------------------------------------------------------
// unv003 Universal Value 03
// ----------------------------------------------------------
// process value to UnV
//      L     0.000000e+000
//      T     "C01UnVD".unv003.ValExt

NETWORK
TITLE =Special Input

      NOP   0;

// ----------------------------------------------------------
// LS_LLL_T13 LS- Tank 13
// ----------------------------------------------------------
      CLR   ;
      =     DB211.DBX   81.4;
      CLR   ;
      =     DB211.DBX   81.5;


// ----------------------------------------------------------
// LS_HL_T13 LS+ Tank 13
// ----------------------------------------------------------
      CLR   ; // Used to stop Filling
      =     DB211.DBX  141.4;
      =     DB211.DBX  141.5;

// ----------------------------------------------------------
// GOA_T13_ML Mannloch Tank 13
// ----------------------------------------------------------
      SET   ;
      =     DB211.DBX  201.4;
      =     DB211.DBX  201.5;

// ----------------------------------------------------------
// U13_SpI04 spare
// ----------------------------------------------------------
      CLR   ;
      =     DB211.DBX  261.4;
      =     DB211.DBX  261.5;

// ----------------------------------------------------------
// LS_LL_T13 LS/ Tank 13
// ----------------------------------------------------------
      CLR   ;
      =     DB211.DBX  321.4;
      CLR   ;
      =     DB211.DBX  321.5;


// ----------------------------------------------------------
// RM_NI_T13_K4_AUF
// ----------------------------------------------------------
      AN    #U.Seq.Step0;
      =     DB211.DBX  381.4;

      AN    #CIP;
      =     DB211.DBX  381.5;


// ----------------------------------------------------------
// RM_NI_T13_K4_ZU
// ----------------------------------------------------------
      AN    #U.Seq.Step0;
      =     DB211.DBX  441.4;

      A     #U.Seq.Step0;
      O     #CIP;
      =     DB211.DBX  441.5;

// ----------------------------------------------------------
// RM_NI_T13_K2
// ----------------------------------------------------------
      AN    #U.Seq.Step0;
      =     DB211.DBX  501.4;

      A     #CIP;
      AN    #U.Seq.Step0;
      =     DB211.DBX  501.5;

// ----------------------------------------------------------
// U13_SpI009 spare
// ----------------------------------------------------------
      CLR   ;
      =     DB211.DBX  561.4;
      =     DB211.DBX  561.5;

// ----------------------------------------------------------
// RM_NI_T13_K3
// ----------------------------------------------------------
      A     #CIP;
      AN    #U.Seq.Step0;
      =     DB211.DBX  621.4;
      SET   ;
      =     DB211.DBX  621.5;

// ----------------------------------------------------------
// LABOR_FREIG_T13 SCHLUESSELSCHALTER LABOR
// ----------------------------------------------------------
      CLR   ;
      =     DB211.DBX  681.4;
      =     DB211.DBX  681.5;

NETWORK
TITLE =Messages

      NOP   0;

// ----------------------------------------------------------
// msg001 Message 01
// ----------------------------------------------------------
      SET   ;
      R     DB217.DBX   80.7;
      =     DB217.DBX   81.4;

      CLR   ;
      =     DB217.DBX   82.7;

// ----------------------------------------------------------
// msg002 Message 02
// ----------------------------------------------------------
      SET   ;
      R     DB217.DBX  140.7;
      =     DB217.DBX  141.4;

      CLR   ;
      =     DB217.DBX  142.7;

NETWORK
TITLE =Sequence organisation

// SFM supply ----------------------------------------------------------------

// analog value to SFM Niveau Tank 13 -----------------------
      L     DB213.DBD  146;
      T     #U.Seq.SFM[17].Val;

// Offset Level
      L     #U.Seq.Prop.Val1;
      L     DB213.DBD  146;
      -R    ;
      T     #U.Seq.SFM[18].Val;

// Offset Level Emptying
      L     DB213.DBD  146;
      T     #U.Seq.SFM[19].Val;


NETWORK
TITLE =Auto / Manual

      SET   ;
      AN    M    122.2;
      JC    MODE;
      AN    M    120.1;

// assign actuator mode
      AN    M    120.1;
      =     DB210.DBX  105.4;
      =     DB210.DBX  185.4;
      =     DB210.DBX  265.4;
      =     DB210.DBX  345.4;
      =     DB210.DBX  425.4;
      =     DB210.DBX  505.4;
      =     DB210.DBX  585.4;
      =     DB210.DBX  665.4;
      =     DB210.DBX  745.4;
      =     DB210.DBX  825.4;
      =     DB210.DBX  905.4;
      =     DB210.DBX  985.4;
      =     DB210.DBX 1065.4;
      =     DB210.DBX 1145.4;
      =     DB210.DBX 1225.4;
      =     DB210.DBX 1305.4;
      =     DB210.DBX 1385.4;
      =     DB210.DBX 1465.4;
      =     DB210.DBX 1545.4;
      =     DB210.DBX 1625.4;
      =     DB210.DBX 1705.4;
      =     DB210.DBX 1785.4;
      =     DB210.DBX 1865.4;
      =     DB210.DBX 1945.4;
      =     DB210.DBX 2025.4;
      =     DB210.DBX 2105.4;
      =     DB210.DBX 2185.4;
      =     DB210.DBX 2265.4;
      =     DB210.DBX 2345.4;
      =     DB210.DBX 2425.4;
      =     DB210.DBX 2505.4;



MODE: SET   ;

      AN    DB211.DBX  678.7;
      O     #CIP;
      =     #LabRel;

NETWORK
TITLE =U13_Act001 spare
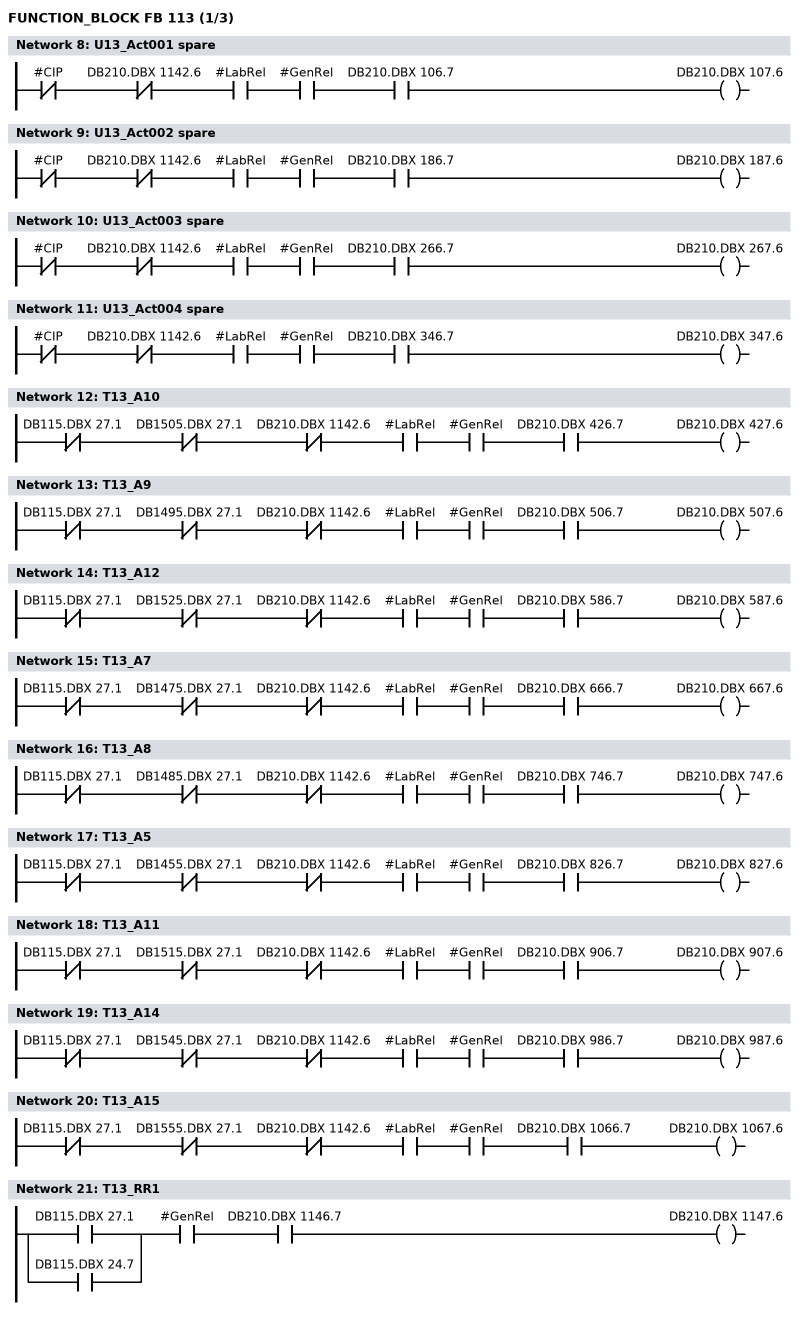

      AN    #CIP;

      AN    DB210.DBX 1142.6;
      A     #LabRel;
      A     #GenRel;
      A     DB210.DBX  106.7;
      =     DB210.DBX  107.6;
NETWORK
TITLE =U13_Act002 spare

      AN    #CIP;

      AN    DB210.DBX 1142.6;
      A     #LabRel;
      A     #GenRel;
      A     DB210.DBX  186.7;
      =     DB210.DBX  187.6;
NETWORK
TITLE =U13_Act003 spare

      AN    #CIP;

      AN    DB210.DBX 1142.6;
      A     #LabRel;
      A     #GenRel;
      A     DB210.DBX  266.7;
      =     DB210.DBX  267.6;
NETWORK
TITLE =U13_Act004 spare

      AN    #CIP;

      AN    DB210.DBX 1142.6;
      A     #LabRel;
      A     #GenRel;
      A     DB210.DBX  346.7;
      =     DB210.DBX  347.6;

NETWORK
TITLE =T13_A10

      AN    DB115.DBX   27.1;
      AN    DB1505.DBX   27.1;

      AN    DB210.DBX 1142.6;
      A     #LabRel;
      A     #GenRel;
      A     DB210.DBX  426.7;
      =     DB210.DBX  427.6;
NETWORK
TITLE =T13_A9

      AN    DB115.DBX   27.1;
      AN    DB1495.DBX   27.1;

      AN    DB210.DBX 1142.6;
      A     #LabRel;
      A     #GenRel;
      A     DB210.DBX  506.7;
      =     DB210.DBX  507.6;
NETWORK
TITLE =T13_A12

      AN    DB115.DBX   27.1;
      AN    DB1525.DBX   27.1;

      AN    DB210.DBX 1142.6;
      A     #LabRel;
      A     #GenRel;
      A     DB210.DBX  586.7;
      =     DB210.DBX  587.6;
NETWORK
TITLE =T13_A7

      AN    DB115.DBX   27.1;
      AN    DB1475.DBX   27.1;

      AN    DB210.DBX 1142.6;
      A     #LabRel;
      A     #GenRel;
      A     DB210.DBX  666.7;
      =     DB210.DBX  667.6;
NETWORK
TITLE =T13_A8

      AN    DB115.DBX   27.1;
      AN    DB1485.DBX   27.1;

      AN    DB210.DBX 1142.6;
      A     #LabRel;
      A     #GenRel;
      A     DB210.DBX  746.7;
      =     DB210.DBX  747.6;
NETWORK
TITLE =T13_A5


      AN    DB115.DBX   27.1;
      AN    DB1455.DBX   27.1;

      AN    DB210.DBX 1142.6;
      A     #LabRel;
      A     #GenRel;
      A     DB210.DBX  826.7;
      =     DB210.DBX  827.6;
NETWORK
TITLE =T13_A11

      AN    DB115.DBX   27.1;
      AN    DB1515.DBX   27.1;

      AN    DB210.DBX 1142.6;
      A     #LabRel;
      A     #GenRel;
      A     DB210.DBX  906.7;
      =     DB210.DBX  907.6;
NETWORK
TITLE =T13_A14

      AN    DB115.DBX   27.1;
      AN    DB1545.DBX   27.1;

      AN    DB210.DBX 1142.6;
      A     #LabRel;
      A     #GenRel;
      A     DB210.DBX  986.7;
      =     DB210.DBX  987.6;

NETWORK
TITLE =T13_A15

      AN    DB115.DBX   27.1;
      AN    DB1555.DBX   27.1;

      AN    DB210.DBX 1142.6;
      A     #LabRel;
      A     #GenRel;
      A     DB210.DBX 1066.7;
      =     DB210.DBX 1067.6;
NETWORK
TITLE =T13_RR1

      A     DB115.DBX   27.1;
      O     DB115.DBX   24.7;
      A     #GenRel;
      A     DB210.DBX 1146.7;
      =     DB210.DBX 1147.6;
NETWORK
TITLE =RV1_T13
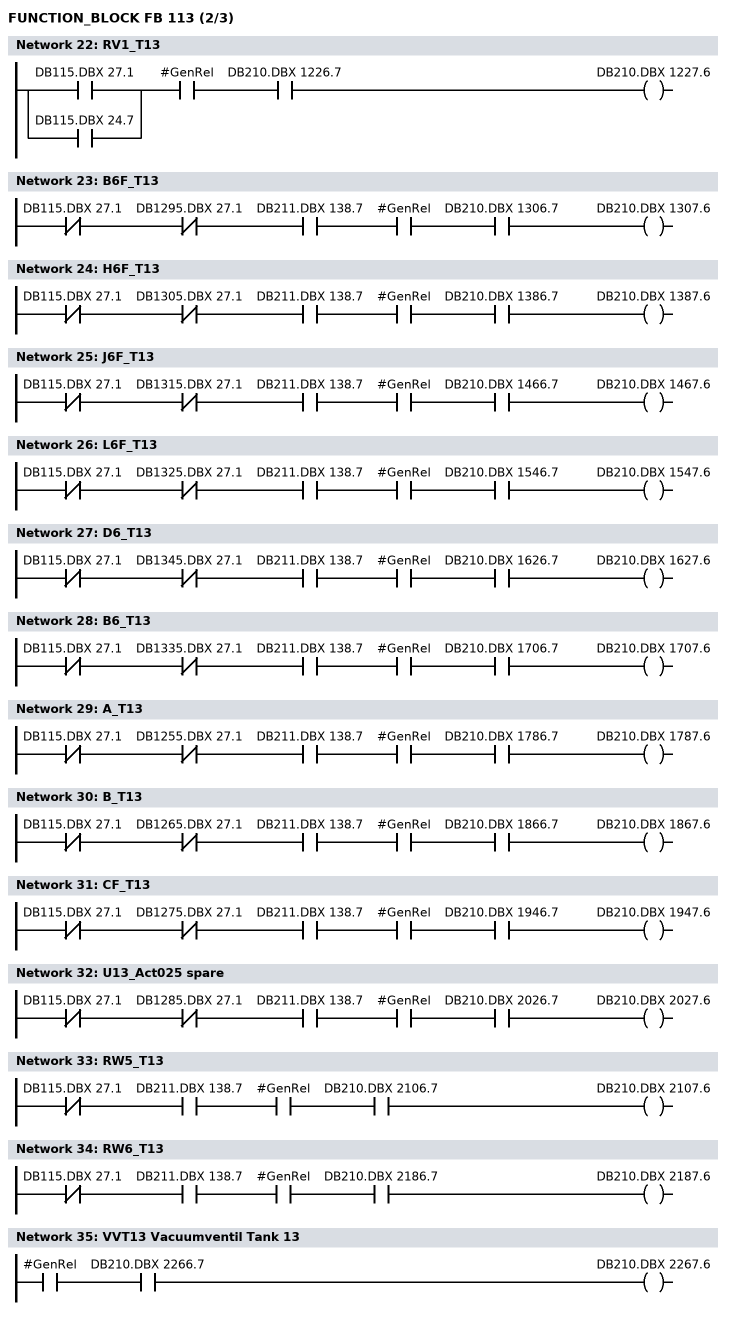

      A     DB115.DBX   27.1;
      O     DB115.DBX   24.7;

      A     #GenRel;
      A     DB210.DBX 1226.7;
      =     DB210.DBX 1227.6;
NETWORK
TITLE =B6F_T13

      AN    DB115.DBX   27.1;
      AN    DB1295.DBX   27.1;

      A     DB211.DBX  138.7;

      A     #GenRel;
      A     DB210.DBX 1306.7;
      =     DB210.DBX 1307.6;
NETWORK
TITLE =H6F_T13

      AN    DB115.DBX   27.1;
      AN    DB1305.DBX   27.1;

      A     DB211.DBX  138.7;

      A     #GenRel;
      A     DB210.DBX 1386.7;
      =     DB210.DBX 1387.6;
NETWORK
TITLE =J6F_T13

      AN    DB115.DBX   27.1;
      AN    DB1315.DBX   27.1;

      A     DB211.DBX  138.7;

      A     #GenRel;
      A     DB210.DBX 1466.7;
      =     DB210.DBX 1467.6;
NETWORK
TITLE =L6F_T13

      AN    DB115.DBX   27.1;
      AN    DB1325.DBX   27.1;

      A     DB211.DBX  138.7;

      A     #GenRel;
      A     DB210.DBX 1546.7;
      =     DB210.DBX 1547.6;
NETWORK
TITLE =D6_T13

      AN    DB115.DBX   27.1;
      AN    DB1345.DBX   27.1;

      A     DB211.DBX  138.7;

      A     #GenRel;
      A     DB210.DBX 1626.7;
      =     DB210.DBX 1627.6;
NETWORK
TITLE =B6_T13

      AN    DB115.DBX   27.1;
      AN    DB1335.DBX   27.1;

      A     DB211.DBX  138.7;

      A     #GenRel;
      A     DB210.DBX 1706.7;
      =     DB210.DBX 1707.6;
NETWORK
TITLE =A_T13

      AN    DB115.DBX   27.1;
      AN    DB1255.DBX   27.1;

      A     DB211.DBX  138.7;

      A     #GenRel;
      A     DB210.DBX 1786.7;
      =     DB210.DBX 1787.6;
NETWORK
TITLE =B_T13

      AN    DB115.DBX   27.1;
      AN    DB1265.DBX   27.1;

      A     DB211.DBX  138.7;

      A     #GenRel;
      A     DB210.DBX 1866.7;
      =     DB210.DBX 1867.6;
NETWORK
TITLE =CF_T13

      AN    DB115.DBX   27.1;
      AN    DB1275.DBX   27.1;

      A     DB211.DBX  138.7;

      A     #GenRel;
      A     DB210.DBX 1946.7;
      =     DB210.DBX 1947.6;
NETWORK
TITLE =U13_Act025 spare

      AN    DB115.DBX   27.1;
      AN    DB1285.DBX   27.1;

      A     DB211.DBX  138.7;

      A     #GenRel;
      A     DB210.DBX 2026.7;
      =     DB210.DBX 2027.6;
NETWORK
TITLE =RW5_T13


      AN    DB115.DBX   27.1;
      A     DB211.DBX  138.7;

      A     #GenRel;
      A     DB210.DBX 2106.7;
      =     DB210.DBX 2107.6;
NETWORK
TITLE =RW6_T13

      AN    DB115.DBX   27.1;
      A     DB211.DBX  138.7;

      A     #GenRel;
      A     DB210.DBX 2186.7;
      =     DB210.DBX 2187.6;
NETWORK
TITLE =VVT13 Vacuumventil Tank 13

      A     #GenRel;
      A     DB210.DBX 2266.7;
      =     DB210.DBX 2267.6;
NETWORK
TITLE =VR_T13
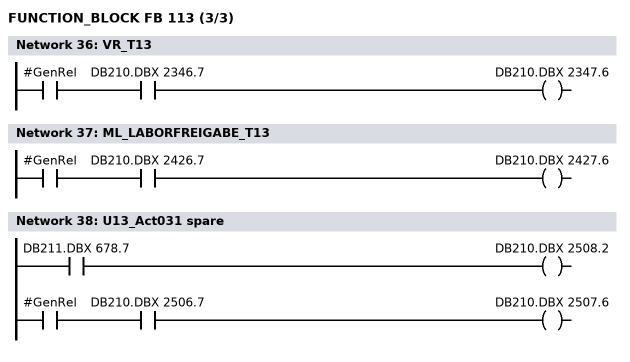

      A     #GenRel;
      A     DB210.DBX 2346.7;
      =     DB210.DBX 2347.6;
NETWORK
TITLE =ML_LABORFREIGABE_T13

      A     #GenRel;
      A     DB210.DBX 2426.7;
      =     DB210.DBX 2427.6;
NETWORK
TITLE =U13_Act031 spare

      A     DB211.DBX  678.7;
      =     DB210.DBX 2508.2;

      A     #GenRel;
      A     DB210.DBX 2506.7;
      =     DB210.DBX 2507.6;
END_FUNCTION_BLOCK

FUNCTION_BLOCK FB 115
TITLE =C01: Water Tank x
AUTHOR : Woermann
FAMILY : BOTEC_F1
NAME : C01Comm
VERSION : 0.1
CODE_VERSION1


VAR
  U : UDT 111;
END_VAR
VAR_TEMP
  iRetVal : INT ;	//return value as integer
  wRetVal : WORD ;	//return value as word
  Run : BOOL ;	//Unit in "RUN" mode
  EStopOK : BOOL ;	//Emergency Stop OK
  CIP : BOOL ;	//CIP Program Selected
  ComCIP : BOOL ;	//Communication with CIP Active
  xTmp : BOOL ;	//Temporary BOOL (free for general use)
  iTmp : INT ;	//Temporary INT (free for general use)
  rTmp : REAL ;	//Temporary REAL (free for general use)
  dTmp : DINT ;	//Temporary DINT (free for general use)
  UnitNo : INT ;	//Unit Number
  EqID : INT ;	//Equipment ID
  Prid : DINT ;	//Process ID
  SFM36 : STRUCT 	//CIP Pump Mode
   I00 : BOOL ;	// Off
   I01 : BOOL ;	// Flow
   I02 : BOOL ;	// Pressure
   I03 : BOOL ;	// Fix Speed
   I04 : BOOL ;
   I05 : BOOL ;
   I06 : BOOL ;
   I07 : BOOL ;
   I08 : BOOL ;
   I09 : BOOL ;
   I10 : BOOL ;
   I11 : BOOL ;
   I12 : BOOL ;
   I13 : BOOL ;
   I14 : BOOL ;
   I15 : BOOL ;
   I16 : BOOL ;
   I17 : BOOL ;
   I18 : BOOL ;
   I19 : BOOL ;
   I20 : BOOL ;
   I21 : BOOL ;
   I22 : BOOL ;
   I23 : BOOL ;
   I24 : BOOL ;
   I25 : BOOL ;
   I26 : BOOL ;
   I27 : BOOL ;
   I28 : BOOL ;
   I29 : BOOL ;
   I30 : BOOL ;
   I31 : BOOL ;
  END_STRUCT ;
  iPLC : INT ;
  iUnit : INT ;
  rUnitNo : REAL ;
  DSTUnit : INT ;	//Destination Unit
  SRCUnit : INT ;
  STBYUnit : INT ;
  rEqID : REAL ;
  dst0 : BOOL ;	//No Destination Selected
  comDST : BOOL ;
END_VAR
BEGIN
NETWORK
TITLE =general

      SET   ;

// unit & equipment number ---------------------------------------------------
      L     #U.Seq.UnitNo;
      T     #UnitNo;

      L     DB115.DBW   14;
      L     1000;
      *I    ;
      L     #UnitNo;
      +I    ;
      T     #EqID;

      L     #EqID;
      ITD   ;
      DTR   ;
      T     #rEqID;


// CIP ----------------------------------------------------------------------
      L     DB115.DBW   18;
      L     0;
      <I    ;
      =     #CIP;

// Communicating Units-------------------------------------------------------
      L     DB115.DBD   10;
      L     DB115.DBD  106;
      ==D   ;
      =     #ComCIP;


NETWORK
TITLE =read other unit's data

      SET   ;

// ... General Unit ----------/

      CALL SFC   20 (
           SRCBLK                   := DB1995.Own,
           RET_VAL                  := #iRetVal,
           DSTBLK                   := DB115.GEN);

// emergency OK -------------------------------------------------------------
      A     DB115.DBX   75.0; //General Emergency Stop OK
      =     #EStopOK;

// ... CIP Unit ------------- /

      CALL SFC   20 (
           SRCBLK                   := DB1915.Own,
           RET_VAL                  := #iRetVal,
           DSTBLK                   := DB115.CIP);



      JU    next;

      L     0;
      T     #iTmp;
      CALL SFC   21 (
           BVAL                     := #iTmp,
           RET_VAL                  := #iRetVal,
           BLK                      := DB115.SRC);


      L     DB1215.DBD   38;
      L     #rEqID;
      ==R   ;
      O(    ;
      L     DB1215.DBD   42;
      L     #rEqID;
      ==R   ;
      )     ;
      O(    ;
      L     DB1215.DBD   46;
      L     #rEqID;
      ==R   ;
      )     ;
      =     #xTmp;

      L     DB1215.DBD   30;
      L     DB115.DBD   30;
      ==R   ;
      O     M    120.7;
      A     #xTmp;
      JCN   N021;
      CALL SFC   20 (
           SRCBLK                   := DB1215.Own,
           RET_VAL                  := #iTmp,
           DSTBLK                   := DB115.SRC);

N021: NOP   0;

next: NOP   0;




















//----------------------------------------
// Communication Well Transfer
//----------------------------------------
      A     #U.Seq.Step0;
      JCN   REM1;
      L     0.000000e+000;
      T     #U.Seq.User.Real1;
REM1: NOP   0;

      L     #U.Seq.User.Real1;
      L     0.000000e+000;
      ==R   ;
      =     #xTmp;

      JCN   CPY1;


// Priority 1
      L     #rEqID;
      L     DB1215.DBD   38;
      ==R   ;
      JCN   U021;
      L     3.021000e+003;
      JU    SRC1;
U021: NOP   0;
      L     #rEqID;
      L     DB1225.DBD   38;
      ==R   ;
      JCN   U022;
      L     3.022000e+003;
      JU    SRC1;
U022: NOP   0;
      L     #rEqID;
      L     DB1255.DBD   38;
      ==R   ;
      JCN   U025;
      L     3.025000e+003;
      JU    SRC1;
U025: NOP   0;
      L     #rEqID;
      L     DB1265.DBD   38;
      ==R   ;
      JCN   U026;
      L     3.026000e+003;
      JU    SRC1;
U026: NOP   0;
      L     #rEqID;
      L     DB1275.DBD   38;
      ==R   ;
      JCN   U027;
      L     3.027000e+003;
      JU    SRC1;
U027: NOP   0;
      L     #rEqID;
      L     DB1285.DBD   38;
      ==R   ;
      JCN   U028;
      L     3.028000e+003;
      JU    SRC1;
U028: NOP   0;
      L     #rEqID;
      L     DB1295.DBD   38;
      ==R   ;
      JCN   U029;
      L     3.029000e+003;
      JU    SRC1;
U029: NOP   0;
      L     #rEqID;
      L     DB1305.DBD   38;
      ==R   ;
      JCN   U030;
      L     3.000000e+001;
      JU    SRC1;
U030: NOP   0;
      L     #rEqID;
      L     DB1315.DBD   38;
      ==R   ;
      JCN   U031;
      L     3.031000e+003;
      JU    SRC1;
U031: NOP   0;
      L     #rEqID;
      L     DB1325.DBD   38;
      ==R   ;
      JCN   U032;
      L     3.032000e+003;
      JU    SRC1;
U032: NOP   0;
      L     #rEqID;
      L     DB1335.DBD   38;
      ==R   ;
      JCN   U033;
      L     3.033000e+003;
      JU    SRC1;
U033: NOP   0;
      L     #rEqID;
      L     DB1345.DBD   38;
      ==R   ;
      JCN   U034;
      L     3.034000e+003;
      JU    SRC1;
U034: NOP   0;


// Priority 2
      L     #rEqID;
      L     DB1215.DBD   42;
      ==R   ;
      JCN   O021;
      L     3.021000e+003;
      JU    SRC1;
O021: NOP   0;
      L     #rEqID;
      L     DB1225.DBD   42;
      ==R   ;
      JCN   O022;
      L     3.022000e+003;
      JU    SRC1;
O022: NOP   0;
      L     #rEqID;
      L     DB1255.DBD   42;
      ==R   ;
      JCN   O025;
      L     3.025000e+003;
      JU    SRC1;
O025: NOP   0;
      L     #rEqID;
      L     DB1265.DBD   42;
      ==R   ;
      JCN   O026;
      L     3.026000e+003;
      JU    SRC1;
O026: NOP   0;
      L     #rEqID;
      L     DB1275.DBD   42;
      ==R   ;
      JCN   O027;
      L     3.027000e+003;
      JU    SRC1;
O027: NOP   0;
      L     #rEqID;
      L     DB1285.DBD   42;
      ==R   ;
      JCN   O028;
      L     3.028000e+003;
      JU    SRC1;
O028: NOP   0;
      L     #rEqID;
      L     DB1295.DBD   42;
      ==R   ;
      JCN   O029;
      L     3.029000e+003;
      JU    SRC1;
O029: NOP   0;
      L     #rEqID;
      L     DB1305.DBD   42;
      ==R   ;
      JCN   O030;
      L     3.000000e+001;
      JU    SRC1;
O030: NOP   0;
      L     #rEqID;
      L     DB1315.DBD   42;
      ==R   ;
      JCN   O031;
      L     3.031000e+003;
      JU    SRC1;
O031: NOP   0;
      L     #rEqID;
      L     DB1325.DBD   42;
      ==R   ;
      JCN   O032;
      L     3.032000e+003;
      JU    SRC1;
O032: NOP   0;
      L     #rEqID;
      L     DB1335.DBD   42;
      ==R   ;
      JCN   O033;
      L     3.033000e+003;
      JU    SRC1;
O033: NOP   0;
      L     #rEqID;
      L     DB1345.DBD   42;
      ==R   ;
      JCN   O034;
      L     3.034000e+003;
      JU    SRC1;
O034: NOP   0;


// Priority 3
      L     #rEqID;
      L     DB1215.DBD   46;
      ==R   ;
      JCN   P021;
      L     3.021000e+003;
      JU    SRC1;
P021: NOP   0;
      L     #rEqID;
      L     DB1225.DBD   46;
      ==R   ;
      JCN   P022;
      L     3.022000e+003;
      JU    SRC1;
P022: NOP   0;
      L     #rEqID;
      L     DB1255.DBD   46;
      ==R   ;
      JCN   P025;
      L     3.025000e+003;
      JU    SRC1;
P025: NOP   0;
      L     #rEqID;
      L     DB1265.DBD   46;
      ==R   ;
      JCN   P026;
      L     3.026000e+003;
      JU    SRC1;
P026: NOP   0;
      L     #rEqID;
      L     DB1275.DBD   46;
      ==R   ;
      JCN   P027;
      L     3.027000e+003;
      JU    SRC1;
P027: NOP   0;
      L     #rEqID;
      L     DB1285.DBD   46;
      ==R   ;
      JCN   P028;
      L     3.028000e+003;
      JU    SRC1;
P028: NOP   0;
      L     #rEqID;
      L     DB1295.DBD   46;
      ==R   ;
      JCN   P029;
      L     3.029000e+003;
      JU    SRC1;
P029: NOP   0;
      L     #rEqID;
      L     DB1305.DBD   46;
      ==R   ;
      JCN   P030;
      L     3.000000e+001;
      JU    SRC1;
P030: NOP   0;
      L     #rEqID;
      L     DB1315.DBD   46;
      ==R   ;
      JCN   P031;
      L     3.031000e+003;
      JU    SRC1;
P031: NOP   0;
      L     #rEqID;
      L     DB1325.DBD   46;
      ==R   ;
      JCN   P032;
      L     3.032000e+003;
      JU    SRC1;
P032: NOP   0;
      L     #rEqID;
      L     DB1335.DBD   46;
      ==R   ;
      JCN   P033;
      L     3.033000e+003;
      JU    SRC1;
P033: NOP   0;
      L     #rEqID;
      L     DB1345.DBD   46;
      ==R   ;
      JCN   P034;
      L     3.034000e+003;
      JU    SRC1;
P034: NOP   0;


      JU    REM2;
SRC1: NOP   0;
      A     #xTmp;
      O     #U.Seq.Step0;
      JCN   REM2;
      T     #U.Seq.User.Real1;
REM2: NOP   0;

      L     #U.Seq.User.Real1;
      L     0.000000e+000;
      >R    ;
      JC    CPY1;
      T     #iTmp;
      CALL SFC   21 (
           BVAL                     := #iTmp,
           RET_VAL                  := #iRetVal,
           BLK                      := DB115.SRC);
      JU    END1;


CPY1: NOP   0;
      CALL FC   950 (
           EquipmentNo              := #U.Seq.User.Real1,
           PLCNo                    := #iPLC,
           UnitNo                   := #iUnit);


      CALL FC   563 (
           ActReq                   := TRUE,
           PLCNo                    := #iPLC,
           SourceUnitNo             := #iUnit,
           IsTUnit                  := FALSE,
           DstComDRec               := DB115.SRC,
           RET_VAL                  := #wRetVal);
END1: NOP   0;

      A     #U.Seq.Step0;
      O     DB115.DBX  219.2;
      L     #U.Seq.User.Real1; // Tank Selection
      L     0.000000e+000;
      >R    ;
      A     DB115.DBX  218.3;
      =     #U.Seq.User.Bit1; // Start Tank

      AN    #U.Seq.Step0;
      R     #U.Seq.User.Bit1; // Start Tank

      L     DB115.DBW  206;
      L     L#1000000;
      *D    ;
      T     #dTmp;

      L     DB115.DBW  208;
      L     1000;
      *D    ;

      L     #dTmp;
      +D    ;
      L     1;
      +D    ;
      NEGD  ;
      T     #U.Seq.User.Dint0;


NETWORK
TITLE =external releases

      SET   ;
      =     DB210.DBX  426.7;
      =     DB210.DBX  506.7;
      =     DB210.DBX  586.7;
      =     DB210.DBX  666.7;
      =     DB210.DBX  746.7;
      =     DB210.DBX  826.7;
      =     DB210.DBX  906.7;
      =     DB210.DBX  986.7;
      =     DB210.DBX 1146.7;
      =     DB210.DBX 1226.7;
      =     DB210.DBX 1306.7;
      =     DB210.DBX 1386.7;
      =     DB210.DBX 1466.7;
      =     DB210.DBX 1546.7;
      =     DB210.DBX 1626.7;
      =     DB210.DBX 1706.7;
      =     DB210.DBX 1786.7;
      =     DB210.DBX 1866.7;
      =     DB210.DBX 1946.7;
      =     DB210.DBX 2106.7;
      =     DB210.DBX 2186.7;
      =     DB210.DBX 2266.7;
      =     DB210.DBX 2346.7;
      =     DB210.DBX 2426.7;
      =     DB210.DBX 2506.7;
NETWORK
TITLE =write own unit data

      SET   ;

//-- CIP Communication ---------------------------------------
      AN    #U.Seq.Step0;
//      AN #U.Seq.PO.B30 // CIP Active (Slave)
      A     #ComCIP;
      JCN   NCIP;
//Conductivity CIP Return
      L     DB115.DBD  150;
      T     #U.Seq.SFM[32].Val;

//Temperature CIP Return
      L     DB115.DBD  146;
      T     #U.Seq.SFM[30].Val;

//CIP Prerun Pump SP
      CALL FC    45 (
           SFM                      := #U.Seq.SFM[36].Sp,
           Indexes                  := #SFM36);


      L     0.000000e+000;
      A     #SFM36.I01;
      =     DB115.DBX  171.7;
      JCN   pfc;
      L     #U.Seq.SFM[34].Sp;
pfc:  NOP   0;
      A     #SFM36.I02;
      =     DB115.DBX  172.0;
      JCN   ppc;
      L     #U.Seq.SFM[35].Sp;
ppc:  NOP   0;
      A     #SFM36.I03;
      =     DB115.DBX  171.6;
      JCN   pxc;
      L     #U.Seq.SFM[29].Sp;
pxc:  NOP   0;
      T     DB115.DBD  182;

// CIP Prerun Temperature
      L     #U.Seq.SFM[36].Sp;
      T     DB115.DBD  182;

//CIP Return
      L     #U.Seq.SFM[28].Sp;
      T     DB115.DBD  186;
      L     DB115.DBD  138;
      T     #U.Seq.SFM[28].Val;

//CIP Prerun
      L     #U.Seq.SFM[27].Sp;
      T     DB115.DBD  190;
      L     DB115.DBD  142;
      T     #U.Seq.SFM[27].Val;

// Write Own Data to CIP
      L     DB115.DBD   10;
      T     DB115.DBD  154;

      L     DB115.DBW   14;
      T     DB115.DBW  158;

      L     DB115.DBW   16;
      T     DB115.DBW  160;

      L     DB115.DBW   18;
      T     DB115.DBW  162;

      L     DB115.DBW   20;
      T     DB115.DBW  164;

      L     DB115.DBW   22;
      T     DB115.DBW  166;

      A     DB115.DBX   24.0;
      =     DB115.DBX  168.0;

      A     DB115.DBX   24.1;
      =     DB115.DBX  168.1;

      A     DB115.DBX   24.2;
      =     DB115.DBX  168.2;

      A     DB115.DBX   24.3;
      =     DB115.DBX  168.3;

      A     DB115.DBX   24.4;
      =     DB115.DBX  168.4;

      A     DB115.DBX   24.5;
      =     DB115.DBX  168.5;

      A     DB115.DBX   24.6;
      =     DB115.DBX  168.6;

      A     DB115.DBX   24.7;
      =     DB115.DBX  168.7;

      L     DB115.DBD  138; // CIP Amount
      T     DB115.DBD   54; // CIP Amount

// Copy Data to CIP
      CALL SFC   20 (
           SRCBLK                   := DB115.ToCIP,
           RET_VAL                  := #iRetVal,
           DSTBLK                   := DB502.ToCIP1);

NCIP: NOP   0;

//Empty Signal
      A     DB211.DBX   78.7;
      =     DB115.DBX   26.5;

//Full Signal
      AN    DB211.DBX  138.7;
      =     DB115.DBX   26.2;

//CIP Program Selected
      A     #CIP;
      =     DB115.DBX   27.1;

// Emergency Stop
      A     #EStopOK; //If needed add or replace with own SpI
      =     DB115.DBX   27.0; //Emergency Stop OK

// Material
      L     #U.Seq.SFM[42].Sp; // Material
      T     DB115.DBD   30;

//----------------------------------------
// Communication Well Transfer
//----------------------------------------
      A     #U.Seq.SFM[18].D; // Level Offset
      AN    DB115.DBX   26.2;
      S     DB115.DBX   27.2;

      AN    #U.Seq.SFM[18].D; // Level Offset
      AN    DB115.DBX   26.0;
      AN    DB115.DBX   26.1;
      O     DB115.DBX   26.2;
      R     DB115.DBX   27.2;

//----------------------------------------
// Communication Water Transfer to Plant
//----------------------------------------
      A     #U.Seq.SFM[19].D; // Empty release
      AN    DB115.DBX   26.5;
      S     DB115.DBX   27.3;

      AN    #U.Seq.SFM[19].D; // Level Offset
      AN    DB115.DBX   26.3;
      AN    DB115.DBX   26.4;
      O     DB115.DBX   26.5;
      R     DB115.DBX   27.3;


NETWORK
TITLE = read from other unit data



END_FUNCTION_BLOCK

FUNCTION_BLOCK FB 119
TITLE =C01: Water Tank x
AUTHOR : Woermann
FAMILY : BOTEC_F1
NAME : C01Sim
VERSION : 0.1
CODE_VERSION1


VAR
  U : UDT 111;
END_VAR
VAR_TEMP
  CIP : BOOL ;	//CIP active
  xTmp : BOOL ;	//Temporary BOOL (free for general use)
  iTmp : INT ;	//Temporary INT (free for general use)
  rTmp : REAL ;	//Temporary REAL (free for general use)
  UnitNo : INT ;	//Unit Number
END_VAR
BEGIN
NETWORK
TITLE =General

      SET   ;
// get unit number ----------------------------------------------------------
      L     #U.Seq.UnitNo;
      T     #UnitNo;

// CIP ----------------------------------------------------------------------
      L     #U.Seq.ProgNo;
      L     0;
      <D    ;
      =     #CIP;

NETWORK
TITLE =Actuator

      A     #U.Seq.Sim;
      =     DB210.DBX  425.3;
      =     DB210.DBX  505.3;
      =     DB210.DBX  665.3;
      =     DB210.DBX  585.3;
      =     DB210.DBX  745.3;
      =     DB210.DBX  825.3;
      =     DB210.DBX  905.3;
      =     DB210.DBX  985.3;
      =     DB210.DBX 1145.3;
      =     DB210.DBX 1225.3;
      =     DB210.DBX 1305.3;
      =     DB210.DBX 1385.3;
      =     DB210.DBX 1465.3;
      =     DB210.DBX 1545.3;
      =     DB210.DBX 1625.3;
      =     DB210.DBX 1705.3;
      =     DB210.DBX 1785.3;
      =     DB210.DBX 1865.3;
      =     DB210.DBX 1945.3;
      =     DB210.DBX 2105.3;
      =     DB210.DBX 2185.3;
      =     DB210.DBX 2265.3;
      =     DB210.DBX 2345.3;
      =     DB210.DBX 2505.3;
      =     DB210.DBX 2425.3;

NETWORK
TITLE =Special Input

      A     #U.Seq.Sim;
      =     DB211.DBX   81.3;
      =     DB211.DBX  141.3;
      =     DB211.DBX  201.3;
      =     DB211.DBX  261.3;
//     =     "WT13SpID".GOA_T13_VV.Sim;
      =     DB211.DBX  381.3;
      =     DB211.DBX  441.3;
      =     DB211.DBX  501.3;
      =     DB211.DBX  621.3;
      =     DB211.DBX  681.3;

NETWORK
TITLE =Counter

      A     #U.Seq.Sim;
      A     M    101.0;
      CLR   ;
NETWORK
TITLE =Analog Input

      A     #U.Seq.Sim;
      =     DB213.DBX  141.3;

NETWORK
TITLE =Universal Value

      A     #U.Seq.Sim;
//      =     "WT13UnVD".unv001.Sim;
//      =     "WT13UnVD".unv002.Sim;
//      =     "WT13UnVD".unv003.Sim;

NETWORK
TITLE =PID

      A     #U.Seq.Sim;

NETWORK
TITLE =Message

      A     #U.Seq.Sim;
//      =     "WT13MsgD".msg001.Sim;
//      =     "WT13MsgD".msg002.Sim;

NETWORK
TITLE =VLT

      A     #U.Seq.Sim;

END_FUNCTION_BLOCK

FUNCTION_BLOCK FB 121
TITLE =C02: Well Transfer x
// NW  1 : phase and index evaluation
// NW  2 : phase  1: start position
// NW  3 : phase  3: Prerinse
// NW  4 : phase  4: Fill System
// NW  5 : phase  5: Transfer
// NW  6 : phase  6: Standby
// NW  7 : phase  8: Push Out
// NW  8 : phase 11: Postrinse
// NW  9 : phase 21: Prepare Line
// NW 10 : phase 22: Tank Selection
// NW 11 : end of sequence
// NW 12 : unit hold request
//SFM   Use                                 Datatype        UoM
//----+-------------------------------------------------------------------------
// 09 : Process Time                        Duration        min
// 40 : Density                             Value           kg/l
// 42 : Material                            Value
// 43 : Destination                         Enumeration
// 44 : Standby                             Val
AUTHOR : Woermann
NAME : C02Seq
VERSION : 0.1
CODE_VERSION1


VAR
  U : UDT 121;
END_VAR
VAR_TEMP
  CIP : BOOL ;	//CIP active
  ComCIP : BOOL ;	//Communication With CIP Active
  ComSRC : BOOL ;	//Communication With Well Managment x
  RRel : BOOL ;	//Run Release
  EStopOK : BOOL ;	//emergency OK
  StepMax : BOOL ;	//StepMax (last) active
  SubStepMax : BOOL ;	//SubStepMax (last) active
  SubStepMaxD : BOOL ;	//SubStepMax (last) done
  ChkOK : BOOL ;	//SubStepMax (last) done
  xTmp : BOOL ;	//Temporary BOOL (free for general use)
  iTmp : INT ;	//Temporary INT (free for general use)
  dTmp : DINT ;	//Temporary DINT (free for general use)
  rTmp : REAL ;	//Temporary REAL (free for general use)
  dUnitNo : DINT ;	//Unit Number
  UnitNo : INT ;	//Unit Number
  EquipmentID : INT ;	//Equipment ID
  S2I : STRUCT 	//SFM to indexes
   SFM26 : STRUCT 	//Cip Step On Condition
    I00 : BOOL ;	//Please Select
    I01 : BOOL ;	//Conductivity High
    I02 : BOOL ;	//Conductivity Low
    I03 : BOOL ;	//Time
    I04 : BOOL ;	//Amount
    I05 : BOOL ;	//Temperature High
    I06 : BOOL ;	//Temperature Low
    I07 : BOOL ;
    I08 : BOOL ;
    I09 : BOOL ;
    I10 : BOOL ;
    I11 : BOOL ;
    I12 : BOOL ;
    I13 : BOOL ;
    I14 : BOOL ;
    I15 : BOOL ;
    I16 : BOOL ;
    I17 : BOOL ;
    I18 : BOOL ;
    I19 : BOOL ;
    I20 : BOOL ;
    I21 : BOOL ;
    I22 : BOOL ;
    I23 : BOOL ;
    I24 : BOOL ;
    I25 : BOOL ;
    I26 : BOOL ;
    I27 : BOOL ;
    I28 : BOOL ;
    I29 : BOOL ;
    I30 : BOOL ;
    I31 : BOOL ;
   END_STRUCT ;
   SFM27 : STRUCT 	//Cip Prerun
    I00 : BOOL ;	//None
    I01 : BOOL ;	//Recovered Water
    I02 : BOOL ;	//Caustic
    I03 : BOOL ;
    I04 : BOOL ;	//Acid
    I05 : BOOL ;
    I06 : BOOL ;
    I07 : BOOL ;
    I08 : BOOL ;
    I09 : BOOL ;
    I10 : BOOL ;
    I11 : BOOL ;
    I12 : BOOL ;	//Fresh Water
    I13 : BOOL ;	//Warm Water
    I14 : BOOL ;
    I15 : BOOL ;
    I16 : BOOL ;
    I17 : BOOL ;
    I18 : BOOL ;
    I19 : BOOL ;
    I20 : BOOL ;
    I21 : BOOL ;
    I22 : BOOL ;
    I23 : BOOL ;
    I24 : BOOL ;
    I25 : BOOL ;
    I26 : BOOL ;
    I27 : BOOL ;
    I28 : BOOL ;
    I29 : BOOL ;
    I30 : BOOL ;
    I31 : BOOL ;
   END_STRUCT ;
   SFM28 : STRUCT 	//Cip Return
    I00 : BOOL ;	//None
    I01 : BOOL ;	//Recovered Water
    I02 : BOOL ;	//Caustic
    I03 : BOOL ;
    I04 : BOOL ;	//Acid
    I05 : BOOL ;
    I06 : BOOL ;
    I07 : BOOL ;
    I08 : BOOL ;
    I09 : BOOL ;
    I10 : BOOL ;
    I11 : BOOL ;
    I12 : BOOL ;	//Fresh Water
    I13 : BOOL ;	//Warm Water
    I14 : BOOL ;
    I15 : BOOL ;	//Drain
    I16 : BOOL ;
    I17 : BOOL ;
    I18 : BOOL ;
    I19 : BOOL ;
    I20 : BOOL ;
    I21 : BOOL ;
    I22 : BOOL ;
    I23 : BOOL ;
    I24 : BOOL ;
    I25 : BOOL ;
    I26 : BOOL ;
    I27 : BOOL ;
    I28 : BOOL ;
    I29 : BOOL ;
    I30 : BOOL ;
    I31 : BOOL ;
   END_STRUCT ;
   SFM37 : STRUCT 	//Cip Pump Mode
    I00 : BOOL ;	//Off
    I01 : BOOL ;	//Flow
    I02 : BOOL ;	//Pressure
    I03 : BOOL ;	//Fix Speed
    I04 : BOOL ;
    I05 : BOOL ;
    I06 : BOOL ;
    I07 : BOOL ;
    I08 : BOOL ;
    I09 : BOOL ;
    I10 : BOOL ;
    I11 : BOOL ;
    I12 : BOOL ;
    I13 : BOOL ;
    I14 : BOOL ;
    I15 : BOOL ;
    I16 : BOOL ;
    I17 : BOOL ;
    I18 : BOOL ;
    I19 : BOOL ;
    I20 : BOOL ;
    I21 : BOOL ;
    I22 : BOOL ;
    I23 : BOOL ;
    I24 : BOOL ;
    I25 : BOOL ;
    I26 : BOOL ;
    I27 : BOOL ;
    I28 : BOOL ;
    I29 : BOOL ;
    I30 : BOOL ;
    I31 : BOOL ;
   END_STRUCT ;
   SFM31 : STRUCT 	//Cip Distribution Circuit No
    I00 : BOOL ;	//Please Select
    I01 : BOOL ;	//Auto Select
    I02 : BOOL ;
    I03 : BOOL ;
    I04 : BOOL ;
    I05 : BOOL ;
    I06 : BOOL ;
    I07 : BOOL ;
    I08 : BOOL ;
    I09 : BOOL ;
    I10 : BOOL ;
    I11 : BOOL ;
    I12 : BOOL ;
    I13 : BOOL ;
    I14 : BOOL ;
    I15 : BOOL ;
    I16 : BOOL ;
    I17 : BOOL ;
    I18 : BOOL ;
    I19 : BOOL ;
    I20 : BOOL ;
    I21 : BOOL ;
    I22 : BOOL ;
    I23 : BOOL ;
    I24 : BOOL ;
    I25 : BOOL ;
    I26 : BOOL ;
    I27 : BOOL ;
    I28 : BOOL ;
    I29 : BOOL ;
    I30 : BOOL ;
    I31 : BOOL ;
   END_STRUCT ;
   SFM39 : STRUCT 	//Q-Status
    I00 : BOOL ;	//Please select
    I01 : BOOL ;	//released
    I02 : BOOL ;
    I03 : BOOL ;
    I04 : BOOL ;
    I05 : BOOL ;
    I06 : BOOL ;	//Ignore
    I07 : BOOL ;
    I08 : BOOL ;
    I09 : BOOL ;	//locked
    I10 : BOOL ;
    I11 : BOOL ;
    I12 : BOOL ;
    I13 : BOOL ;
    I14 : BOOL ;
    I15 : BOOL ;
    I16 : BOOL ;
    I17 : BOOL ;
    I18 : BOOL ;
    I19 : BOOL ;
    I20 : BOOL ;
    I21 : BOOL ;
    I22 : BOOL ;
    I23 : BOOL ;
    I24 : BOOL ;
    I25 : BOOL ;
    I26 : BOOL ;
    I27 : BOOL ;
    I28 : BOOL ;
    I29 : BOOL ;
    I30 : BOOL ;
    I31 : BOOL ;
   END_STRUCT ;
   SFM10 : STRUCT 	//Current Tank
    I00 : BOOL ;	//Please Select
    I01 : BOOL ;	//Water Tank 1
    I02 : BOOL ;	//Water Tank 2
    I03 : BOOL ;	//Water Tank 2
    I04 : BOOL ;	//Water Tank 3
    I05 : BOOL ;	//Water Tank 4
    I06 : BOOL ;	//Water Tank 5
    I07 : BOOL ;	//Water Tank 6
    I08 : BOOL ;	//Water Tank 7
    I09 : BOOL ;	//Water Tank 8
    I10 : BOOL ;	//WAter Tank 9
    I11 : BOOL ;	//Water Tank 10
    I12 : BOOL ;	//Water Tank 11
    I13 : BOOL ;	//Water Tank 12
    I14 : BOOL ;	//Water Tank 13
    I15 : BOOL ;
    I16 : BOOL ;
    I17 : BOOL ;
    I18 : BOOL ;
    I19 : BOOL ;
    I20 : BOOL ;
    I21 : BOOL ;
    I22 : BOOL ;
    I23 : BOOL ;
    I24 : BOOL ;
    I25 : BOOL ;
    I26 : BOOL ;
    I27 : BOOL ;
    I28 : BOOL ;
    I29 : BOOL ;
    I30 : BOOL ;
    I31 : BOOL ;
   END_STRUCT ;
   SFM11 : STRUCT 	//1. Tank
    I00 : BOOL ;	//Please Select
    I01 : BOOL ;	//Water Tank 1
    I02 : BOOL ;	//Water Tank 2
    I03 : BOOL ;	//Water Tank 2
    I04 : BOOL ;	//Water Tank 3
    I05 : BOOL ;	//Water Tank 4
    I06 : BOOL ;	//Water Tank 5
    I07 : BOOL ;	//Water Tank 6
    I08 : BOOL ;	//Water Tank 7
    I09 : BOOL ;	//Water Tank 8
    I10 : BOOL ;	//WAter Tank 9
    I11 : BOOL ;	//Water Tank 10
    I12 : BOOL ;	//Water Tank 11
    I13 : BOOL ;	//Water Tank 12
    I14 : BOOL ;	//Water Tank 13
    I15 : BOOL ;
    I16 : BOOL ;
    I17 : BOOL ;
    I18 : BOOL ;
    I19 : BOOL ;
    I20 : BOOL ;
    I21 : BOOL ;
    I22 : BOOL ;
    I23 : BOOL ;
    I24 : BOOL ;
    I25 : BOOL ;
    I26 : BOOL ;
    I27 : BOOL ;
    I28 : BOOL ;
    I29 : BOOL ;
    I30 : BOOL ;
    I31 : BOOL ;
   END_STRUCT ;
   SFM12 : STRUCT 	//2. Tank
    I00 : BOOL ;	//Please Select
    I01 : BOOL ;	//Water Tank 1
    I02 : BOOL ;	//Water Tank 2
    I03 : BOOL ;	//Water Tank 2
    I04 : BOOL ;	//Water Tank 3
    I05 : BOOL ;	//Water Tank 4
    I06 : BOOL ;	//Water Tank 5
    I07 : BOOL ;	//Water Tank 6
    I08 : BOOL ;	//Water Tank 7
    I09 : BOOL ;	//Water Tank 8
    I10 : BOOL ;	//WAter Tank 9
    I11 : BOOL ;	//Water Tank 10
    I12 : BOOL ;	//Water Tank 11
    I13 : BOOL ;	//Water Tank 12
    I14 : BOOL ;	//Water Tank 13
    I15 : BOOL ;
    I16 : BOOL ;
    I17 : BOOL ;
    I18 : BOOL ;
    I19 : BOOL ;
    I20 : BOOL ;
    I21 : BOOL ;
    I22 : BOOL ;
    I23 : BOOL ;
    I24 : BOOL ;
    I25 : BOOL ;
    I26 : BOOL ;
    I27 : BOOL ;
    I28 : BOOL ;
    I29 : BOOL ;
    I30 : BOOL ;
    I31 : BOOL ;
   END_STRUCT ;
   SFM13 : STRUCT 	//3. Tank
    I00 : BOOL ;	//Please Select
    I01 : BOOL ;	//Water Tank 1
    I02 : BOOL ;	//Water Tank 2
    I03 : BOOL ;	//Water Tank 2
    I04 : BOOL ;	//Water Tank 3
    I05 : BOOL ;	//Water Tank 4
    I06 : BOOL ;	//Water Tank 5
    I07 : BOOL ;	//Water Tank 6
    I08 : BOOL ;	//Water Tank 7
    I09 : BOOL ;	//Water Tank 8
    I10 : BOOL ;	//WAter Tank 9
    I11 : BOOL ;	//Water Tank 10
    I12 : BOOL ;	//Water Tank 11
    I13 : BOOL ;	//Water Tank 12
    I14 : BOOL ;	//Water Tank 13
    I15 : BOOL ;
    I16 : BOOL ;
    I17 : BOOL ;
    I18 : BOOL ;
    I19 : BOOL ;
    I20 : BOOL ;
    I21 : BOOL ;
    I22 : BOOL ;
    I23 : BOOL ;
    I24 : BOOL ;
    I25 : BOOL ;
    I26 : BOOL ;
    I27 : BOOL ;
    I28 : BOOL ;
    I29 : BOOL ;
    I30 : BOOL ;
    I31 : BOOL ;
   END_STRUCT ;
  END_STRUCT ;
  ComCIPDist : BOOL ;	//Communication with CIP Distribution
  ComDST : BOOL ;	//Communication with Water Tank
  ComWT1 : BOOL ;	//Comminication with unit Water Treatment 1 OK
  FLT : BOOL ;	//Line has Carbon Filter
  rUnitNo : REAL ;	//Unit Number Real
  CurrSel : REAL ;	//Current Tank Selection SP
  ComWTank2 : BOOL ;	//Communication Water Tank Priority 2
  ComWTank3 : BOOL ;	//Communication Water Tank Priority 3
  ComWTank1 : BOOL ;	//Communication Water Tank Priority 1
  ComPLN : BOOL ;	//Communication with Transfer Plan
END_VAR
BEGIN
NETWORK
TITLE = Phase and Index Evaluation

      CLR   ;
      =     #RRel;

// ---------------------------------------------------------------------------
// write max used SFM's (last SFM number + 1)
      L     46;
      T     #U.SFMQuant;

// ---------------------------------------------------------------------------
// unit & equipment number
      L     MB   112;
      T     #UnitNo;

      L     DB125.DBW   14;
      L     1000;
      *I    ;
      L     #UnitNo;
      +I    ;
      T     #EquipmentID;

// ---------------------------------------------------------------------------
// CIP active
      L     MW   114;
      L     0;
      <I    ;
      =     #CIP;

// ---------------------------------------------------------------------------
// communicating units
      L     MD   124;
      L     DB125.DBD  106;
      ==D   ;
      =     #ComCIP;

      L     MD   124;
      L     DB125.DBD  202;
      ==D   ;
      =     #ComSRC;

      L     DB125.DBD  318; // Destination Material
      L     #U.Seq.SFM[42].Sp;
      ==R   ;
      =     #ComDST;

      L     DB125.DBD  366; // Destination Material
      L     #U.Seq.SFM[42].Sp;
      ==R   ;
      =     #ComWTank1;

      L     DB125.DBD  414; // Destination Material
      L     #U.Seq.SFM[42].Sp;
      ==R   ;
      =     #ComWTank2;

      L     DB125.DBD  462; // Destination Material
      L     #U.Seq.SFM[42].Sp;
      ==R   ;
      =     #ComWTank3;


// Load Source to SFM
      L     DB125.DBD  242;
      T     #U.Seq.SFM[14].Sp;


// ---------------------------------------------------------------------------
// process timer start
      SET   ;
      =     M    131.0;

// ---------------------------------------------------------------------------
// emergency OK
      A     DB125.DBX   27.0;
      =     #EStopOK;

// define last (Sub)Step active
      L     #U.Seq.StepMax;
      L     MW   104;
      ==I   ;
      =     #StepMax;

      L     #U.Seq.SubStepMax;
      L     MW   118;
      ==I   ;
      =     #SubStepMax;

      A     #SubStepMax;
      A     #U.Seq.SPD;
      AN    M    103.2;
      =     #SubStepMaxD;

// ---------------------------------------------------------------------------
// index evaluation: Current Tank
      CALL FC    45 (
           SFM                      := #U.Seq.SFM[10].Sp,
           Indexes                  := #S2I.SFM10);

// index evaluation: 1. Tank
      CALL FC    45 (
           SFM                      := #U.Seq.SFM[11].Sp,
           Indexes                  := #S2I.SFM11);

// index evaluation: 2. Tank
      CALL FC    45 (
           SFM                      := #U.Seq.SFM[12].Sp,
           Indexes                  := #S2I.SFM12);

// index evaluation: 3. Tank
      CALL FC    45 (
           SFM                      := #U.Seq.SFM[13].Sp,
           Indexes                  := #S2I.SFM13);

// index evaluation: Q-Status
      CALL FC    45 (
           SFM                      := #U.Seq.SFM[39].Sp,
           Indexes                  := #S2I.SFM39);

// ---------------------------------------------------------------------------
// phase evaluation
      L     MW   108;
      JL    X0;
      JU    X0; // phase  0:
      JU    X1; // phase  1: start position
      JU    X0; // phase  2:
      JU    X3; // phase  3: Prerinse
      JU    X4; // phase  4: Fill System
      JU    X5; // phase  5: Transfer
      JU    X6; // phase  6: Standby
      JU    X0; // phase  7:
      JU    X8; // phase  8: Push Out
      JU    X0; // phase  9:
      JU    X0; // phase 10:
      JU    X11; // phase 11: Postrinse
      JU    X0; // phase 12:
      JU    X0; // phase 13:
      JU    X0; // phase 14:
      JU    X0; // phase 15:
      JU    X0; // phase 16:
      JU    X0; // phase 17:
      JU    X0; // phase 18:
      JU    X0; // phase 19:
      JU    X0; // phase 20:
      JU    X21; // phase 21: Prepare Line
      JU    X22; // phase 22: Tank Selection
X0:   SET   ;
      S     M    108.7; // Error unknown phase
      JU    COMM;
NETWORK
TITLE =phase 1: startposition

X1:   SET   ;
// ---------------------------------------------------------------------------
// general functions
// ---------------------------------------------------------------------------
// reset signals
      A     M    102.2;
      R     #U.Seq.Switch.Sw1;
      R     #U.Seq.Switch.Sw2;
      R     DB125.DBX   26.1;

      L     0.000000e+000;
      T     DB125.DBD   30;
      T     DB125.DBD   34;
      T     DB125.DBD   38;
      T     DB125.DBD   42;
      T     DB125.DBD   46;
      T     DB125.DBD   50;
      T     DB125.DBD   54;
      T     #U.Seq.SFM[10].Sp;
      T     #U.Seq.SFM[11].Sp;
      T     #U.Seq.SFM[12].Sp;
      T     #U.Seq.SFM[13].Sp;

      AN    M    102.0;
      =     M    161.0; // Reset Process Timer

      CALL FC   709 (// Reset "Simulation" And "Ignore"
           UnitNo                   := #UnitNo,// Of All Control Modules
           Enable                   := M    102.2);// At First Cycle of Startposition (Idle)

// ---------------------------------------------------------------------------
// start check --------------------------------------------------------------
      A     #CIP;
      JC    M010;

      CALL FC   120 (
           ChkType                  := 1,// production
           ChkOK                    := M    122.0);
      JU    COMM;

M010: CALL FC   120 (
           ChkType                  := 2,// CIP
           ChkOK                    := M    122.0);
      JU    COMM;
NETWORK
TITLE =phase 3: Prerinse
//SFM   Use                                 Datatype        UoM
//----+-------------------------------------------------------------------------
// 00 : Watch Dog Time                      Duration        min
// 20 : Flow                                Value           l/h
// 41 : Amount                              Value           kg
X3:   SET   ;
// ---------------------------------------------------------------------------
// General CM evaluation
      CALL FC   120 (
           ChkType                  := 3,
           ChkOK                    := #ChkOK);

      AN    #ChkOK;
      S     M    120.3;

// ---------------------------------------------------------------------------
// general functions
      AN    M    121.2;
      A     M    102.3;
      =     #RRel;

      CALL FC   779 (
           P1Sel                    := #U.Seq.SFM[11].Sp,
           P2Sel                    := #U.Seq.SFM[12].Sp,
           P3Sel                    := #U.Seq.SFM[13].Sp,
           P1Rel                    := DB125.DBX  363.2,
           P2Rel                    := DB125.DBX  411.2,
           P3Rel                    := DB125.DBX  459.2,
           CurrSel                  := #U.Seq.User.Real10);

      L     #U.Seq.User.Real10;
      T     #U.Seq.SFM[10].Sp;

// ---------------------------------------------------------------------------
// messages
      A     #S2I.SFM39.I01; // Released
      JCN   N301;
      L     919; // "Press Start to Continue"
      T     MD    90;
N301: NOP   0;

      A     M    151.6; // Rinse Amount
      A     #S2I.SFM39.I00; // Please Select
      JCN   N302;
      L     816; // LAB Release Required
      T     MD    90;
N302: NOP   0;

// ---------------------------------------------------------------------------
// timer & counter
      A     M    102.0;
      =     M    131.6;

// Presinse
      AN    #U.Seq.SFM[15].P;
      =     #xTmp;
      CALL FC   710 (
           RefVal                   := DB125.DBD  230,
           Active                   := #xTmp,
           Reset                    := #U.Seq.SFM[15].Res,
           Down                     := FALSE,
           CntVal                   := #U.Seq.SFM[15].Val,
           RefMem                   := #U.Seq.User.Real1);

// ---------------------------------------------------------------------------
// pause timer  .
      SET   ;
      S     M    141.7;
// ---------------------------------------------------------------------------
// communication
// Water Tank
      A     M    102.3;
      =     DB125.DBX   26.3;


// Well Management
      A     DB220.DBX  102.6;
      AN    M    151.6; // Rinse Amount
      A     M    102.3;
      =     DB125.DBX   26.1; // Request Water


// ---------------------------------------------------------------------------
// Check Partner
      AN    #ComSRC;
      O(    ;
      AN    DB125.DBX  218.3;
      AN    DB125.DBX  218.4;
      )     ;
      AN    #U.Seq.Step0;
      AN    #CIP;
      JCN   NC03;
      L     904; // "Source Not Ready!
      T     MD    90;
NC03: NOP   0;

      AN    DB125.DBX  314.0; // Water Tank Ready
      AN    DB125.DBX  314.1;
      AN    #ComDST;
      A     #S2I.SFM10.I00;
      AN    #U.Seq.Step0;
      AN    #U.Seq.PO.B22;
      AN    #CIP;
      JCN   NC04;
      L     903; // Destination not Ready
      T     MD    90;
NC04: NOP   0;

// ---------------------------------------------------------------------------
// control modules
// Drain
      A     #ComSRC; // Coms Well Management
      A     DB125.DBX   75.2;
      AN    M    151.6;
      A     M    102.3;
      =     DB220.DBX  108.0;

// CO2
//      A     "C02ComD".DST.Fill
//      A     #ComDST
      L     #U.Seq.SFM[22].Sp;
      L     1.000000e+001;
      <R    ;
      A(    ;
      L     #U.Seq.SFM[22].Sp;
      L     5.000000e+000;
      >R    ;
      )     ;
      A     DB125.DBX  218.4;
      A     DB125.DBX  219.7;
      A     M    103.3;
      =     DB220.DBX  348.0;
      =     DB220.DBX  188.0;
      =     DB220.DBX  268.0;

